METHOD PUBLIC initJntPos : BOOL
VAR_INPUT
END_VAR
m_lastLinkEncoder :=m_motorInputs.m_linkEncoder;
m_linkEncCycles:=0;
m_curLinkPos :=linkEnc2Pos();
m_initLinkPos:=m_curLinkPos;
m_initMotorEnc :=m_motorInputs.m_motorEncoder;
m_curMotorPos:=motorEnc2Pos();
m_curJntPos := m_curMotorPos;
m_cmdJntPos :=m_curJntPos;	
m_lastJntPos :=m_curJntPos;
m_lastLinkPos := m_curLinkPos;

// filter init
m_jntVelLpf.init(1, g_curJntVelLpfCutoffFreq, g_armCtrlFreq);
m_linkVelLpf.init(1, g_curJntVelLpfCutoffFreq, g_armCtrlFreq);
END_METHOD

// reset the initial joint position with input value
METHOD PUBLIC initJntPosReset : BOOL
VAR_INPUT
	i_initLinkPos:LREAL;
END_VAR
m_initLinkPos:=i_initLinkPos;
m_initMotorEnc :=m_motorInputs.m_motorEncoder;
m_curMotorPos:=motorEnc2Pos();
m_curJntPos := m_curMotorPos;
m_cmdJntPos :=m_curJntPos;	
m_lastJntPos :=m_curJntPos;
m_lastLinkPos := m_curLinkPos;

// filter init
m_jntVelLpf.init(1, g_curJntVelLpfCutoffFreq, g_armCtrlFreq);
m_linkVelLpf.init(1, g_curJntVelLpfCutoffFreq, g_armCtrlFreq);
END_METHOD

PROPERTY initLinkPos : lreal
GET
initLinkPos:=m_initLinkPos;
END_GET
SET
m_initLinkPos:=initLinkPos;
END_SET
END_PROPERTY

METHOD PUBLIC isEnabled : BOOL
VAR_INPUT
END_VAR
isEnabled :=(DriverStatusWord_OP = m_motorInputs.m_statusWord);
END_METHOD

PROPERTY jntPos : LREAL
GET
jntPos := m_curJntPos;
END_GET
END_PROPERTY

PROPERTY jntTrq : LREAL
GET
jntTrq:=m_curJntTrq;
END_GET
END_PROPERTY

PROPERTY jntVel : LREAL
GET
jntVel := m_curJntVel;
END_GET
END_PROPERTY

METHOD PROTECTED linkEnc2Pos : LREAL
VAR_INPUT
END_VAR
VAR
	incLinkPos :LREAL;
	newLinkEnc :DINT;
END_VAR
// cycle check
IF 1=m_multiCycles THEN
	IF (m_motorInputs.m_linkEncoder - m_lastLinkEncoder)*m_linkEncoderDir < -m_linkEncoderRes/2 THEN
		m_linkEncCycles :=m_linkEncCycles+1;
	ELSIF (m_motorInputs.m_linkEncoder - m_lastLinkEncoder)*m_linkEncoderDir > m_linkEncoderRes/2 THEN
		m_linkEncCycles :=m_linkEncCycles-1;
	END_IF
END_IF
m_lastLinkEncoder:=m_motorInputs.m_linkEncoder;

// convert link encoder if joint cross zero
newLinkEnc := m_motorInputs.m_linkEncoder;
IF 1=m_linkEncZeroCross AND 0 = m_multiCycles THEN
	IF 1=m_linkEncoderDir AND m_motorInputs.m_linkEncoder < m_minLinkEncoder THEN
		newLinkEnc := m_motorInputs.m_linkEncoder + m_linkEncoderRes;
	ELSIF -1=m_linkEncoderDir AND m_motorInputs.m_linkEncoder < m_maxLinkEncoder THEN
		newLinkEnc := m_motorInputs.m_linkEncoder + m_linkEncoderRes;
	END_IF
END_IF

// motion from calibrated points
incLinkPos := (newLinkEnc-m_caliLinkEncoder)*m_linkEnc2PosRatio;

// absolute joint position
linkEnc2Pos := incLinkPos + m_linkEncCaliJntPos + 2*PI* m_linkEncCycles;
END_METHOD

PROPERTY PUBLIC linkPos : LREAL
GET
linkPos:=m_curLinkPos;
END_GET
END_PROPERTY

METHOD PROTECTED motorEnc2Pos : LREAL
VAR_INPUT
END_VAR
motorEnc2Pos:= (m_motorInputs.m_motorEncoder-m_initMotorEnc)* m_motorEnc2PosRatio +m_initLinkPos;
END_METHOD

PROPERTY PUBLIC motorPos : LREAL
GET
motorPos := m_curMotorPos;
END_GET
END_PROPERTY

METHOD PROTECTED motorPos2Enc : DINT
VAR_INPUT
	i_jntPos :LREAL;
END_VAR

VAR
END_VAR
motorPos2Enc := LREAL_TO_DINT((i_jntPos-m_initLinkPos)/m_motorEnc2PosRatio + m_initMotorEnc);
END_METHOD

PROPERTY rawCurrent : LREAL
GET
rawCurrent := m_rawCurrent;
END_GET
END_PROPERTY

METHOD PUBLIC updateCmds : BOOL
VAR_INPUT
	i_opMode : E_DriverOPMode;
	i_cmdPos :LREAL;
	i_cmdTrq :LREAL;
END_VAR
VAR
	filtCmdTrq :LREAL;
END_VAR
m_motorOutputs.m_opMode:=INT_TO_SINT( i_opMode);
// pos mode
IF i_opMode = DriverOPMode_Pos THEN
	m_motorOutputs.m_cmdCurrent:=0;
	m_cmdTrqLpf.reset();
//	i_cmdPos:=LIMIT(m_minJntPos, i_cmdPos, m_maxJntPos);
	m_motorOutputs.m_cmdMotorEncoder :=motorPos2Enc(i_cmdPos);
ELSIF i_opMode = DriverOPMode_Trq THEN
	filtCmdTrq:=m_cmdTrqLpf.run(i_cmdTrq);
	m_motorOutputs.m_cmdCurrent:=LREAL_TO_DINT(LIMIT(-m_maxCurrent, filtCmdTrq*m_trq2CurrentRatio,m_maxCurrent));
	m_motorOutputs.m_cmdMotorEncoder :=m_motorInputs.m_motorEncoder; 
END_IF
m_cmdCurrent:=m_motorOutputs.m_cmdCurrent;
END_METHOD

METHOD PUBLIC updateStatus : BOOL
VAR_INPUT
END_VAR
// compute joint position
m_curLinkPos:= linkEnc2Pos();
m_curMotorPos:=motorEnc2Pos();
m_curJntPos := m_curMotorPos;

// compute joint velocity
m_curJntVel:= (m_curJntPos-m_lastJntPos)/m_cycleTime;
m_curJntVel := m_jntVelLpf.run(m_curJntVel);
m_lastJntPos :=m_curJntPos;

// compute link velocity
m_curLinkVel := (m_curLinkPos-m_lastLinkPos)/m_cycleTime;
m_curLinkVel := m_linkVelLpf.run(m_curLinkVel);
m_lastLinkPos := m_curLinkPos;

//compute joint acceleration
m_curJntAcc:=(m_curJntVel-m_lastJntVel)/m_cycleTime;
m_curJntAcc := m_jntAccLpf.run(m_curJntAcc);
m_lastJntVel:=m_curJntVel;

//compute link acceleration
m_curLinkAcc:=(m_curLinkVel-m_lastLinkVel)/m_cycleTime;
m_curLinkAcc := m_linkAccLpf.run(m_curLinkAcc);
m_lastLinkVel:=m_curLinkVel;

// current and torque
m_rawCurrent := m_motorInputs.m_current;
m_filtCurrent := m_curTrqLpf.run(m_rawCurrent);
m_curJntTrq := m_filtCurrent * m_current2TrqRatio;
END_METHOD

END_FUNCTION_BLOCK

// ---- FBs_RobotDynamics/FB_MasterFriciton.TcPOU
FUNCTION_BLOCK FB_MasterFriciton
VAR_INPUT
END_VAR
VAR_OUTPUT
END_VAR
VAR
	// joint friction compensation scale
	m_frictionCompScale :Vec7d :=[0.7, 0.5, 0.5, 0.0, 0.7, 0.7, 0.7];
	
	// joint velocity threshold for coulomb friction transition
	m_cFrictionVelThres : LREAL := 5.0 * g_deg2Rad;
	
	// arm index
	m_armIdx: INT ;
	
	// joint coulomb friction parameters: friction = a * gravityTrq + b;
	m_frictionParamA : Vec7d := g_zeroVec7d;
	m_frictionParamB : Vec7d := g_zeroVec7d;
	
	// joint damping
	m_jntDamp :Vec7d := g_zeroVec7d;
	
	// max joint friciton 
	m_maxFriction :Vec7d;
	

END_VAR

METHOD init : BOOL
VAR_INPUT
	i_armIdx :INT;
END_VAR

VAR
	i:int;
END_VAR
m_armIdx := i_armIdx;

m_frictionParamA := g_zeroVec7d;
m_frictionParamB := g_zeroVec7d;
m_jntDamp := g_zeroVec7d;
m_maxFriction := GVL_ArmDynamics.g_maxJntFriction;

FOR i:=1 TO 7 DO
	m_frictionParamA[i] := GVL_ArmDynamics.g_jntFrictionParam[m_armIdx, 2*i-1];
	m_frictionParamB[i] := GVL_ArmDynamics.g_jntFrictionParam[m_armIdx, 2*i];
END_FOR
END_METHOD

METHOD run : vec7d
VAR_IN_OUT CONSTANT
	// joint gravity torque
	i_jntGravity :Vec7d;
	
	// joint velocity
	i_jntVel :Vec7d;
END_VAR

VAR
	i:INT;
	transitScale:LREAL;
	cFriction, dFriction :LREAL;
END_VAR
FOR i:=1 TO g_mJntNum DO
	transitScale := LIMIT(0, ABS(i_jntVel[i]/m_cFrictionVelThres),1);
	cFriction:=m_frictionParamA[i]*ABS(i_jntGravity[i])+m_frictionParamB[i];
	cFriction:= transitScale * sign(i_jntVel[i]) * cFriction;
	
	dFriction:= i_jntVel[i] * m_jntDamp[i];
	
	run[i] := LIMIT(-m_maxFriction[i], m_frictionCompScale[i] * (cFriction+dFriction) ,m_maxFriction[i]);
END_FOR
END_METHOD

END_FUNCTION_BLOCK

// ---- FBs_Robots/FB_CartJoint.TcPOU
FUNCTION_BLOCK FB_CartJoint EXTENDS FB_JointBase
VAR_INPUT
END_VAR
VAR_OUTPUT
END_VAR
VAR
END_VAR

METHOD PUBLIC init : BOOL
VAR_INPUT
	i_jntIdx :INT;
	i_controlCycleTime :LREAL;
END_VAR
m_cycleTime := i_controlCycleTime;

// hardware parameters
m_motorEncoderRes :=GVL_CartJointParameters.g_incEncoderRes[i_jntIdx];
m_linkEncoderRes :=GVL_CartJointParameters.g_absEncoderRes[i_jntIdx];
m_motorReduction :=GVL_CartJointParameters.g_motorReduction[i_jntIdx];
m_linkEncoderReduction :=GVL_CartJointParameters.g_absEncoderReduction[i_jntIdx];
m_trqConst :=GVL_CartJointParameters.g_motorTrqConst[i_jntIdx];
m_maxCurrent :=GVL_CartJointParameters.g_motorMaxCurrent[i_jntIdx];
m_motorDir :=GVL_CartJointParameters.g_motorDir[i_jntIdx];								
m_linkEncoderDir :=GVL_CartJointParameters.g_asbEncoderDir[i_jntIdx];
m_minJntPos	:=GVL_CartJointParameters.g_minJntPos[i_jntIdx];
m_maxJntPos	:=GVL_CartJointParameters.g_maxJntPos[i_jntIdx];

//link encoder calibartion data
m_minLinkEncoder :=GVL_CartJointCaliData.g_minLinkEncoder[i_jntIdx] - m_linkEncoderDir*GVL_CartJointCaliData.g_linkEncLimitBuffer; // expand limit
m_maxLinkEncoder :=GVL_CartJointCaliData.g_maxLinkEncoder[ i_jntIdx] + m_linkEncoderDir*GVL_CartJointCaliData.g_linkEncLimitBuffer; // expand limit
m_caliLinkEncoder :=GVL_CartJointCaliData.g_caliLinkEncoder[i_jntIdx];
m_linkEncCaliJntPos :=GVL_CartJointCaliData.g_linkEncCaliJntPos[i_jntIdx];
m_linkEncZeroCross :=GVL_CartJointCaliData.g_linkEncZeroCross[i_jntIdx];
m_multiCycles :=GVL_CartJointCaliData.g_multipleCyclesJoint[i_jntIdx];

// convert cali link encoder if joint cross zero
IF 1=m_linkEncZeroCross THEN
	IF 1=m_linkEncoderDir AND m_caliLinkEncoder < m_minLinkEncoder THEN
		m_caliLinkEncoder := GVL_CartJointCaliData.g_caliLinkEncoder[i_jntIdx] + m_linkEncoderRes;
	ELSIF -1=m_linkEncoderDir AND m_caliLinkEncoder < m_maxLinkEncoder THEN
		m_caliLinkEncoder := GVL_CartJointCaliData.g_caliLinkEncoder[i_jntIdx] + m_linkEncoderRes;
	END_IF
END_IF

// macro data
m_trq2CurrentRatio:=m_motorDir * 1000.0/(m_trqConst*m_motorReduction);
m_current2TrqRatio:=m_motorDir * (m_trqConst*m_motorReduction)/1000.0;
m_linkEnc2PosRatio := 2*PI*m_linkEncoderDir/(m_linkEncoderReduction*m_linkEncoderRes);
m_motorEnc2PosRatio := 2*PI * m_motorDir/(m_motorReduction * m_motorEncoderRes);

// motor data init
m_curJntVel:=0;
m_curJntTrq :=0;
m_rawCurrent :=0;
m_filtCurrent :=0;
m_cmdJntVel :=0.0;
m_cmdJntTrq :=0.0;
m_cmdCurrent := 0.0;

// filter init
m_cmdTrqLpf.init(1, g_cmdJntTrqLpfCutoffFreq, g_cartCtrlFreq);
m_curTrqLpf.init(1, g_curJntTrqLpfCutoffFreq, g_cartCtrlFreq);
m_jntVelLpf.init(1, g_curJntVelLpfCutoffFreq, g_cartCtrlFreq);
m_linkVelLpf.init(1, g_curJntVelLpfCutoffFreq, g_cartCtrlFreq);
m_jntAccLpf.init(1, g_curJntVelLpfCutoffFreq*0.2, g_armCtrlFreq); 
m_linkAccLpf.init(1, g_curJntVelLpfCutoffFreq*0.2, g_armCtrlFreq); 


// driver init value
m_motorOutputs.m_controlWord:=DriverCtrlWord_INIT;
m_motorOutputs.m_opMode:=INT_TO_SINT(DriverOPMode_Pos);
m_motorOutputs.m_cmdCurrent:=0;
m_motorOutputs.m_cmdMotorEncoder:=m_motorInputs.m_motorEncoder;
END_METHOD

END_FUNCTION_BLOCK

// ---- FBs_Robots/FB_MasterCart.TcPOU
FUNCTION_BLOCK FB_MasterCart
VAR
	//  IO and check
	m_endoScopePedalIO AT%I* :BOOL;
	m_endoScopeIOCheck :FB_IOCheck;
	
	m_clutchPedalIO AT%I* :BOOL;
	m_clutchIOCheck :FB_IOCheck;
	
	m_surgonHeadInIO AT%I* :BOOL;
	m_headInCheck:FB_IOCheck;
	
	m_armSwitchIO AT%I* :BOOL;
	m_armSwitchCheck:FB_IOToggleCheck;
	
	m_electricCutLeft AT %I* :BOOL;
	m_electricCutLeftAllow AT %I* :BOOL;
	
	m_electricCutRight AT %I* :BOOL;
	m_electricCutRightAllow AT %I* :BOOL;
	
	m_electricCoagulLeft AT %I* :BOOL;
	m_electricCoagulLeftAllow AT %I* :BOOL;
	
	m_electricCoagulRight AT %I* :BOOL;
	m_electricCoagulRightAllow AT %I* :BOOL;
	
	m_elecKnifeCtrlWord AT %Q* :DINT;
	
	// cart status
	m_cartStatus  : ST_CartStatus;
	
	// cart joints
	// [monitor lift, monitor rotate, armset, pedal]
	m_cartJoints:ARRAY[1..4] OF FB_CartJoint;
	
	// cart joint motion control IO
	//[monitor_up, monitor_down, monitor_cwRotate, monitor_ccwRotate, armset_up, armset_down, pedal_in, pedal_out]
	m_cartJointCtrlIO AT%I* :ARRAY[1..8] OF BOOL ;
	m_cartJointCtrlIOCheck :ARRAY[1..8] OF FB_IOCheck;
	
	//electrotome control io
	m_electricCutLeftOn :BOOL;
	m_electricCutRightOn :BOOL;
	m_electricCoagulLeftOn : BOOL;
	m_electricCoagulRightOn : BOOL;
	//Triggering several energies at once
	m_eleCtrlState : UINT;
	//The type of instrument energy of the master hand corresponding to the slave hand
	m_energyType :ARRAY[1..g_mArmNum] OF UINT :=[2(0)];
	
	// cart joint control data
	m_jntEnableCounts:Vec4i ;
	m_jntDisableCounts:Vec4i ;
	m_jntEnableCountsThres:INT:=500;
	m_jntCmdMotionDir :Vec4i;
	m_cmdJntTrq :Vec4d;
	m_cmdJntPos :Vec4d;
	m_cmdJntVel :Vec4d;
	m_jntEnableFlag :Vec4b;
	
	//cart ergonomic adjust data
	m_UIData : ST_CartUIData;
	m_carInMotion : INT; // 0:  no mition, 1: mamual adjust, 2: ergonomic adjust
	m_jntSoftwareLimit :ARRAY [1..4] OF LREAL := [0.001, 1*g_deg2Rad, 0.001, 0.001];
	m_cmdArrival : Vec4b;
	
	// cart joint status data
	m_curMotorPos :Vec4d;
	m_curLinkPos :Vec4d;
	m_curJntPos :Vec4d;
	m_curJntVel :Vec4d;
	m_curJntTrq :Vec4d;
	m_rawJntCurrent :Vec4d;
	m_filtJntCurrent :Vec4d;
	m_cmdJntCurrent : Vec4d;

END_VAR

METHOD eleKnifeCtrl : DINT
VAR_IN_OUT CONSTANT
	m_armState:ARRAY[1..g_mArmNum] OF E_masterArmState ;
	m_teleSlaveArmIdx :ARRAY[1..g_mArmNum] OF E_MatchedSlaveArmIdx;
	m_instruStauts: ARRAY[1..g_sArmNum] OF ST_InstruStatus;
END_VAR
//Foot trigger check
m_electricCutLeftOn := m_electricCutLeft AND m_electricCutLeftAllow AND m_armState[1] = MasterArmState_MasterSlave ;
m_electricCutRightOn := m_electricCutRight AND m_electricCutRightAllow AND m_armState[2] = MasterArmState_MasterSlave ;
m_electricCoagulLeftOn := m_electricCoagulLeft AND m_electricCoagulLeftAllow AND m_armState[1] = MasterArmState_MasterSlave ;
m_electricCoagulRightOn := m_electricCoagulRight AND m_electricCoagulRightAllow AND m_armState[2] = MasterArmState_MasterSlave ;

//You cannot excite two energies at the same time
m_eleCtrlState := BOOL_TO_UINT(m_electricCutLeftOn) + BOOL_TO_UINT(m_electricCutRightOn)
										 + BOOL_TO_UINT(m_electricCoagulLeftOn) + BOOL_TO_UINT(m_electricCoagulRightOn);

IF m_teleSlaveArmIdx[1] > 0 THEN
	m_energyType[1] := m_instruStauts[m_teleSlaveArmIdx[1]].m_energyType;
	m_energyType[2] := m_instruStauts[m_teleSlaveArmIdx[2]].m_energyType;
END_IF

IF m_eleCtrlState = 1 THEN
	IF (m_electricCutLeftOn AND  m_energyType[1] = InstruType_isMonopole) OR (m_electricCutRightOn AND  m_energyType[2] = InstruType_isMonopole) THEN
		eleKnifeCtrl := EnergyCtrlWord_isMonopoleCut;
	ELSIF (m_electricCoagulLeftOn AND m_energyType[1] = InstruType_isMonopole) OR (m_electricCoagulRightOn AND  m_energyType[2] = InstruType_isMonopole) THEN
		eleKnifeCtrl := EnergyCtrlWord_isMonopoleCoagul;
	ELSIF (m_electricCoagulLeftOn AND m_energyType[1] = InstruType_isBipolar) OR (m_electricCoagulRightOn AND  m_energyType[2] = InstruType_isBipolar) THEN
		eleKnifeCtrl := EnergyCtrlWord_isBipolarCoagul;
	ELSIF (m_electricCutLeftOn AND m_energyType[1] = InstruType_isUltraKnife) OR (m_electricCutRightOn AND  m_energyType[2] = InstruType_isUltraKnife) THEN
		eleKnifeCtrl := EnergyCtrlWord_isUltraMin;
	ELSIF (m_electricCoagulLeftOn AND m_energyType[1] = InstruType_isUltraKnife) OR (m_electricCoagulRightOn AND  m_energyType[2] = InstruType_isUltraKnife) THEN
		eleKnifeCtrl := EnergyCtrlWord_isUltraMax;
		
	ELSE
		eleKnifeCtrl := EnergyCtrlWord_NoOutput;
	END_IF
ELSE
	eleKnifeCtrl := EnergyCtrlWord_NoOutput;
END_IF
END_METHOD

METHOD ergonomicAdjust : INT
VAR_INPUT
END_VAR
VAR
	i : INT;
	err:Vec4d;
END_VAR
vecSub(m_UIData.m_cmdJntPos,m_curJntPos, err);
ergonomicAdjust := 2;
//only update command after joints is truly enabled
FOR i := 1 TO 4 DO
	IF m_jntEnableFlag[i] AND m_cartJoints[i].isEnabled() AND m_jntEnableCounts[i]>= m_jntEnableCountsThres THEN
		m_cmdJntVel[i]:=sign(m_UIData.m_cmdJntPos[i]-m_cartJoints[i].jntPos)*(GVL_CartJointParameters.g_jntCtrlMotionVel[i]);
		IF ABS(err[i]) < m_jntSoftwareLimit[i]/3 THEN
			m_cmdJntVel[i]:=0;
		END_IF
		m_cmdJntPos[i] := LIMIT(GVL_CartJointParameters.g_minJntPos[i] + m_jntSoftwareLimit[i],  m_cmdJntPos[i] + m_cmdJntVel[i]*g_cartCtrlCycleTime, GVL_CartJointParameters.g_maxJntPos[i] - m_jntSoftwareLimit[i]);
	
	ELSE
		m_cmdJntVel[i]:=0;
		m_cmdJntPos[i] := m_cartJoints[i].jntPos;
	END_IF	
END_FOR
END_METHOD

METHOD PUBLIC getStatus : BOOL
VAR_IN_OUT
	// cart status data
	r_cartStatus :ST_CartStatus;
	
	// cart joint data
	r_cartJointData :ST_CartJointData;
	
END_VAR
r_cartStatus := m_cartStatus;


// current joint data
r_cartJointData.m_curMotorPos:=m_curMotorPos;
r_cartJointData.m_curLinkPos:=m_curLinkPos;
r_cartJointData.m_curJntPos:=m_curJntPos;
r_cartJointData.m_curJntVel:=m_curJntVel;
r_cartJointData.m_curJntTrq:=m_curJntVel;
r_cartJointData.m_rawJntCurrent:=m_rawJntCurrent;
r_cartJointData.m_filtJntCurrent:=m_filtJntCurrent;

// command joint data
r_cartJointData.m_cmdJntPos:=m_cmdJntPos;
r_cartJointData.m_cmdJntVel:=m_cmdJntVel;
r_cartJointData.m_cmdJntTrq:=m_cmdJntTrq;
r_cartJointData.m_cmdJntCurrent:=m_cmdJntCurrent;
END_METHOD

METHOD PUBLIC init : BOOL
VAR_INPUT
END_VAR
VAR
	i:INT;
	initLinkPos :LREAl;
END_VAR
// joint init
FOR i:=1 TO 4 DO
	m_cartJoints[i].init(i,g_cartCtrlCycleTime);
	m_cartJoints[i].initJntPos();
END_FOR

// motor and link encoder of  monitor rotation are on different  joints
// transfer monitor angle from link side to motor side
initLinkPos:= monitorAngLink2Motor(m_cartJoints[2].initLinkPos);
m_cartJoints[2].initJntPosReset(initLinkPos);

// init commands
FOR i:=1 TO 4 DO
	m_jntEnableCounts[i]:=0;
	m_jntDisableCounts[i]:=0;
	m_jntEnableFlag[i]:=FALSE;
	m_jntCmdMotionDir[i]:=0;
	m_cmdJntTrq[i]:=0;
	m_cmdJntVel[i]:=0;
	m_cmdJntPos[i]:=m_cartJoints[i].jntPos;
END_FOR

m_cartStatus.m_initFlag :=true;
END_METHOD

METHOD manualAdjust : INT
VAR_INPUT
END_VAR
VAR
	i : INT;
END_VAR
// update joint command positon
manualAdjust := 1;
//only update command after joints is truly enabled
FOR i := 1 TO 4 DO
	IF  m_jntEnableFlag[i] AND m_cartJoints[i].isEnabled() AND m_jntEnableCounts[i]>= m_jntEnableCountsThres THEN
		//  update command joint velocity
		m_cmdJntVel[i]:=m_jntCmdMotionDir[i]*GVL_CartJointParameters.g_jntCtrlMotionVel[i];
		
		// limit handle
		IF (m_cmdJntPos[i]> GVL_CartJointParameters.g_maxJntPos[i] - m_jntSoftwareLimit[i] AND m_cmdJntVel[i] >0 ) OR 
				(m_cmdJntPos[i]< GVL_CartJointParameters.g_minJntPos[i] + m_jntSoftwareLimit[i] AND m_cmdJntVel[i] <0 )  THEN
				m_cmdJntVel[i] := 0.0;
		END_IF
		m_cmdJntPos[i]:= m_cmdJntPos[i]+ m_cmdJntVel[i]*g_cartCtrlCycleTime;
	ELSE
		m_cmdJntVel[i]:=0;
		m_cmdJntPos[i] := m_cartJoints[i].jntPos;
	END_IF
END_FOR
END_METHOD

// TODO
METHOD PROTECTED monitorAngLink2Image : LREAL
VAR_INPUT
	i_linkPos:LREAL;
END_VAR
VAR
	A,B,C,D,E,F,G,H,I,X0,X1,X2,X3,X4,X5,X6,X7,X8,X9,X10,X11,X12,Z0:LREAL;	
END_VAR

X0:=i_linkPos;  //监视器旋转

A:=227; B:=216; C:=159.285; D:=150.297; E:=195; F:=130; G:=137; H:=40; I:=99;
X4:=ATAN(H/I); X5:=ATAN(F/G);
X8:=SQRT(F*F+G*G);
X12:=sqrt(H*H+I*I);
X9:=sqrt(E*E+X12*X12-2*E*X12*cos(X0));
X6:=acos((B*B+X8*X8-X9*X9)/(2*B*X8));
X10:=acos((B*B+X9*X9-X8*X8)/(2*B*X9));
X11:=acos((X9*X9+X12*X12-E*E)/(2*X9*X12));
X7:=X10+X11;
X2:=X5-X6;
X3:=pi-X7+X2;
X1:=X3-X4;

monitorAngLink2Image:=X1;
END_METHOD

// TODO
METHOD PROTECTED monitorAngLink2Motor : LREAL
VAR_INPUT
	i_linkPos:LREAL;
END_VAR
VAR
	A,B,C,D,E,F,G,H,I,X0,X1,X2,X3,X4,X5,X6,X7,X8,X9,X10,X11,X12,Z0:LREAL;	
END_VAR

X0:=i_linkPos;  //监视器旋转

A:=227; B:=216; C:=159.285; D:=150.297; E:=195; F:=130; G:=137; H:=40; I:=99;
X4:=ATAN(H/I); X5:=ATAN(F/G);
X8:=SQRT(F*F+G*G);
X12:=sqrt(H*H+I*I);
X9:=sqrt(E*E+X12*X12-2*E*X12*cos(X0));
X6:=acos((B*B+X8*X8-X9*X9)/(2*B*X8));
X10:=acos((B*B+X9*X9-X8*X8)/(2*B*X9));
X11:=acos((X9*X9+X12*X12-E*E)/(2*X9*X12));
X7:=X10+X11;
X2:=X5-X6;
X3:=pi-X7+X2;
X1:=X3-X4;

monitorAngLink2Motor:=X2;
END_METHOD

//TODO
METHOD PROTECTED monitorAngMotor2Link : LREAL
VAR_INPUT
	i_motorPos:LREAL;
END_VAR
VAR
	A,B,C,D,E,F,G,H,I,X0,X1,X2,X3,X4,X5,X6,X7,X8,X9,X10,X11,X12,Z0:LREAL;	
END_VAR
X2:=i_motorPos;

A:=227; B:=216; C:=159.285; D:=150.297; E:=195; F:=130; G:=137; H:=40; I:=99;
X5:=atan(F/G);
X6:=X5-X2;
X8:=sqrt(F*F+G*G);
X9:=sqrt(B*B+X8*X8-2*B*X8*cos(X6));
X12:=SQRT(H*H+I*I);
X0:=ACOS((E*E+X12*X12-X9*X9)/(2*E*X12));

monitorAngMotor2Link:=X0;
END_METHOD

METHOD reachUITargetCheck : bool
VAR
	i :INT;
	err:Vec4d;
END_VAR
vecSub(m_UIData.m_cmdJntPos,m_curJntPos, err);

// joint error check
FOR i:=1 TO 4 DO 
	m_cmdArrival[i] :=  ABS(err[i]) < m_jntSoftwareLimit[i]/2;
END_FOR
END_METHOD

METHOD PUBLIC run : BOOL
VAR_IN_OUT CONSTANT
	i_cartUIData : ST_CartUIData;
END_VAR
VAR
	i:INT;
END_VAR
// update IO signals
updateIO(i_cartUIData);

// update cart status
updateStatus();

// update controller and command
updateCmds();

// send command to joint driver
FOR i:=1 TO 4 DO
	// joint enable
	IF m_jntEnableFlag[i] AND NOT(SafetyCheck.m_safetyCheckData.m_cartErrFlag[i]) AND MasterArmControl.m_masterStatus.m_armState[1] <> MasterArmState_MasterSlave 
								AND MasterArmControl.m_masterStatus.m_armState[2] <> MasterArmState_MasterSlave THEN
		m_cartJoints[i].enable();
	ELSE
		m_cartJoints[i].disable();
	END_IF
	
	// set command position
	m_cartJoints[i].updateCmds(DriverOPMode_Pos,m_cmdJntPos[i],m_cmdJntTrq[i]);
END_FOR
END_METHOD

PROPERTY status : ST_CartStatus
GET
status := m_cartStatus;
END_GET
END_PROPERTY

METHOD PROTECTED updateCmds : BOOL
VAR_INPUT
END_VAR
VAR
	i:INT;
	
END_VAR
IF (m_jntCmdMotionDir[1] <>0 OR m_jntCmdMotionDir[2]<>0 OR m_jntCmdMotionDir[3] <>0 OR m_jntCmdMotionDir[4] <>0) AND m_carInMotion <> 2 THEN
	m_carInMotion := manualAdjust();
ELSIF (m_UIData.m_ergonomicCrl.m_recovErgonEnable OR m_UIData.m_ergonomicCrl.m_cancelRecovErgonEnable) AND m_carInMotion <> 1 THEN
	m_carInMotion := ergonomicAdjust();
ELSE
	m_carInMotion := 0;
END_IF

reachUITargetCheck();
IF m_cmdArrival[1] AND m_cmdArrival[2] AND m_cmdArrival[3] AND m_cmdArrival[4] THEN
	IF m_UIData.m_ergonomicCrl.m_recovErgonEnable THEN
		m_cartStatus.m_cancelErgonAdjustArrival := FALSE;
		m_cartStatus.m_ergonAdjustArrival := TRUE;
	END_IF
	IF m_UIData.m_ergonomicCrl.m_cancelRecovErgonEnable THEN
		m_cartStatus.m_ergonAdjustArrival := FALSE;
		m_cartStatus.m_cancelErgonAdjustArrival := TRUE;
	END_IF
ELSE
	m_cartStatus.m_ergonAdjustArrival := FALSE;
	IF m_UIData.m_ergonomicCrl.m_recovErgonEnable THEN
		m_cartStatus.m_cancelErgonAdjustArrival := FALSE;
	END_IF
END_IF
END_METHOD

METHOD PROTECTED updateIO : BOOL
VAR_INPUT
	i_cartUIData : ST_CartUIData;
END_VAR
VAR
	i:INT;
	idxOffset:INT;
END_VAR
// updata IO signals
m_cartStatus.m_clutchSwitch:= m_clutchIOCheck.check(m_clutchPedalIO);
m_cartStatus.m_endoscopeSwitch := m_endoScopeIOCheck.check(m_endoScopePedalIO);
m_cartStatus.m_surgonReady := m_headInCheck.check(m_surgonHeadInIO);
m_cartStatus.m_armSwitch :=m_armSwitchCheck.check(m_armSwitchIO);
m_UIData := i_cartUIData;

//updata Electrotome control
m_elecKnifeCtrlWord := eleKnifeCtrl(MasterArmControl.m_masterStatus.m_armState , MasterArmControl.m_masterStatus.m_teleSlaveArmIdx , MasterArmControl.m_masterInputDataPool.m_slaveStatus.m_instruStauts );

//updata pedal hover and pedal trigger
m_cartStatus. m_pedalHover[1] := m_electricCutLeftAllow OR m_electricCoagulLeftAllow;
m_cartStatus. m_pedalHover[2] := m_electricCutRightAllow OR m_electricCoagulRightAllow;
IF m_electricCutLeftOn AND m_eleCtrlState = 1 THEN
	m_cartStatus.m_electricKnifePedalTrigger[1] := 1;
ELSIF m_electricCoagulLeftOn AND m_eleCtrlState = 1 THEN
	m_cartStatus.m_electricKnifePedalTrigger[1] := 2;
ELSE
	m_cartStatus.m_electricKnifePedalTrigger[1] := 0;
END_IF

IF m_electricCutRightOn AND m_eleCtrlState = 1 THEN
	m_cartStatus.m_electricKnifePedalTrigger[2] := 1;
ELSIF m_electricCoagulRightOn AND m_eleCtrlState = 1 THEN
	m_cartStatus.m_electricKnifePedalTrigger[2] := 2;
ELSE
	m_cartStatus.m_electricKnifePedalTrigger[2] := 0;
END_IF

//update cart joint control switch
FOR i:=1 TO 4 DO 
	idxOffset:= 2*(i-1);
	IF m_cartJointCtrlIOCheck[1+idxOffset].check(m_cartJointCtrlIO[1+idxOffset]) THEN
		m_jntCmdMotionDir[i]:=1;
	ELSIF  m_cartJointCtrlIOCheck[2+idxOffset].check(m_cartJointCtrlIO[2+idxOffset]) THEN
		m_jntCmdMotionDir[i]:=-1;
	ELSE
		m_jntCmdMotionDir[i]:=0;
	END_IF
END_FOR


// if console is already in motion, only check the currently moving joint
IF m_cartStatus.m_consoleInAdjust THEN
	FOR i:=1 TO 4 DO
		IF NOT(m_cartJoints[i].isEnabled()) THEN
			m_jntCmdMotionDir[i] := 0;
		END_IF
	END_FOR
END_IF


// update joint enable flag
FOR i:= 1 TO 4 DO
	IF m_jntCmdMotionDir[i] <> 0 OR m_UIData.m_ergonomicCrl.m_recovErgonEnable OR m_UIData.m_ergonomicCrl.m_cancelRecovErgonEnable THEN
		m_jntEnableFlag[i] := TRUE;
		m_jntEnableCounts[i]:= LIMIT(0, m_jntEnableCounts[i]+1, m_jntEnableCountsThres);
		m_jntDisableCounts[i]:=m_jntEnableCountsThres;
	ELSE
		m_jntEnableCounts[i]:=0;
		m_jntDisableCounts[i]:= LIMIT(0, m_jntDisableCounts[i]-1, m_jntEnableCountsThres);
		m_jntEnableFlag[i] :=m_jntDisableCounts[i]>0; 
	END_IF
END_FOR

// Do not adjust during master-slave control
IF MasterArmControl.m_masterStatus.m_armState[1] = MasterArmState_MasterSlave OR MasterArmControl.m_masterStatus.m_armState[1] = MasterArmState_Endoscope OR
	MasterArmControl.m_masterStatus.m_armState[2] = MasterArmState_MasterSlave OR MasterArmControl.m_masterStatus.m_armState[2] = MasterArmState_Endoscope  THEN
	m_jntCmdMotionDir := g_zeroVec4i;
END_IF
END_METHOD

METHOD PROTECTED updateStatus : BOOL
VAR_INPUT
END_VAR
VAR
	i:INT;
END_VAR
// update cart joints status
FOR i:=1  TO 4 DO
	m_cartJoints[i].updateStatus();
END_FOR

// get joint data
FOR i:=1 TO 4 DO
	m_curMotorPos[i]:=m_cartJoints[i].motorPos;
	m_curLinkPos[i]:=m_cartJoints[i].linkPos;
	m_curJntPos[i]:=m_cartJoints[i].jntPos;
	m_curJntVel[i]:=m_cartJoints[i].jntVel;
	m_curJntTrq[i]:=m_cartJoints[i].jntTrq;
	m_rawJntCurrent[i]:=m_cartJoints[i].rawCurrent;
	m_filtJntCurrent[i]:=m_cartJoints[i].filtCurrent;
	m_cmdJntCurrent[i]:=m_cartJoints[i].cmdCurrent;
END_FOR 

// transfer monitor angle from link side to motor side
m_curLinkPos[2]:= monitorAngLink2Motor(m_cartJoints[2].linkPos);

// get monitor angle
m_cartStatus.m_monitorAngle:= monitorAngLink2Image(m_cartJoints[2].linkPos);

// check if cart in motion
m_cartStatus.m_consoleInAdjust:=FALSE;
FOR i:=1 TO 4 DO
	IF m_cartJoints[i].isEnabled() THEN
		m_cartStatus.m_consoleInAdjust:=TRUE;
		EXIT;
	END_IF
END_FOR

// check if monitor in motion
m_cartStatus.m_monitorInAdjust:=m_cartJoints[2].isEnabled();

// check if cart in manual adjustment
m_cartStatus.m_consoleInManualAdjust := FALSE;
FOR i:=1 TO 4 DO
	IF m_jntCmdMotionDir[i] <> 0 AND m_cartJoints[i].isEnabled() THEN
		m_cartStatus.m_consoleInManualAdjust := TRUE;
		EXIT;
	END_IF
END_FOR
END_METHOD

END_FUNCTION_BLOCK

// ---- Mains/MasterArmControl.TcPOU
PROGRAM MasterArmControl
VAR
	// slave robot data, input from slave controller box
	m_slaveRobotData AT %I* : MSCommu_slaveStatus;
	
	// all data from other tasks and controller 
	m_masterInputDataPool : ST_MasterInputDataPool;
	
	// master robot information, including arm status and cartesian data, output to other tasks
	m_masterStatus AT %Q* :ST_MasterStatus;
	
	// master robot joint data, output to other tasks
	m_masterJointsData AT %Q* :ST_MasterJointData;
		
	// master robot data, ouput to slave controller box
	m_masterRobotData AT %Q* :MSCommu_MasterStatus;
	
	// flag to init robot
	m_robotInit :BOOL :=FALSE;
	
	// wait time before robot init  for ethercat to be statble 
	m_robotInitWaitTime : LREAL:=0;
	
	// master robot
	m_masterRobot:FB_MasterRobot;
	
	// code execute time measure
	m_codeTime : Profiler;
	
END_VAR

m_codeTime(START:=TRUE, RESET:=TRUE);

// wait communication to be stable
IF(m_robotInitWaitTime<g_robotInitWaitTime) THEN
	m_robotInitWaitTime := m_robotInitWaitTime+g_armCtrlCycleTime;
	RETURN;
END_IF

// robot init
IF m_robotInit =FALSE THEN
	m_masterRobot.Init();
	m_robotInit:=TRUE;
END_IF

// input from UI
UIInputProcess();

// slave input data cast
slaveInputDataCast(m_slaveRobotData, m_masterInputDataPool.m_slaveStatus);

// robot run
m_masterRobot.run(m_masterInputDataPool);

// update data pool
m_masterRobot.getStatus(m_masterStatus,m_masterJointsData);

// master output data cast
masterOutputDataCast(m_masterRobot.m_shoulderPoseInMonitor, m_masterStatus, m_masterRobotData);

// output to UI
UIOutputProcess();

m_codeTime(START:=FALSE);

// convert from local ST_MasterStatus for control to MSCommu_MasterStatus for master-slave communication
METHOD masterOutputDataCast : BOOL
VAR_IN_OUT CONSTANT
	shoulderPose :ARRAY[1..2] OF ST_Frame;
	masterStatus :ST_MasterStatus;
END_VAR
VAR_IN_OUT
	masterOutputData:MSCommu_MasterStatus;
END_VAR

VAR
	i,j : INT;
	poseInMonitor:ST_Frame;
	velInShoulder, wVelInShoulder :Vec3d;
	velInMonitor, wVelInMonitor :Vec3d;
END_VAR
// Master heart beat
IF masterOutputData.m_heartBeat >= 10 THEN
	masterOutputData.m_heartBeat := 0;
ELSE
	masterOutputData.m_heartBeat := masterOutputData.m_heartBeat + 1;
END_IF

masterOutputData.m_motionScale :=masterStatus.m_motionScale;
masterOutputData.m_slaveSelfCheckFlag := m_masterInputDataPool.m_UIData.m_selfCheckFlag;
masterOutputData.m_pedalHover := m_masterInputDataPool.m_cartStatus.m_pedalHover;
masterOutputData.m_electricKnifePedalTrigger := m_masterInputDataPool.m_cartStatus.m_electricKnifePedalTrigger;
masterOutputData.m_tryMSControl[1] := BOOL_TO_INT(m_masterInputDataPool.m_cartStatus.m_surgonReady);
masterOutputData.m_tryMSControl[2] := BOOL_TO_INT(m_masterInputDataPool.m_cartStatus.m_surgonReady);
masterOutputData.m_uiResetFault := GVL_interactUI.g_uiResetFault;
masterOutputData.m_masterStopButton := NOT SafetyCheck.m_stopButton;

FOR i:=1 TO g_mArmNum DO
	masterOutputData.m_armState[i] := masterStatus.m_armState[i];
	masterOutputData.m_teleSlaveArmIdx[i] :=masterStatus.m_teleSlaveArmIdx[i];
	masterOutputData.m_gripAngle[i] := masterStatus.m_gripAngle[i] ;
	
	poseInMonitor := transform(shoulderPose[i],  masterStatus.m_curArmPose[i]);
	masterOutputData.m_curArmPose[i].m_pos := poseInMonitor.m_pos ;
	masterOutputData.m_curArmPose[i].m_rot := poseInMonitor.m_rot ;
	
	FOR j:=1 TO 3 DO
		velInShoulder[j]:=masterStatus.m_curArmTwist[i][j];
		wVelInShoulder[j]:=masterStatus.m_curArmTwist[i][j+3];
	END_FOR
	matMultiVec(shoulderPose[i].m_rot, velInShoulder,velInMonitor);
	matMultiVec(shoulderPose[i].m_rot, wVelInShoulder,wVelInMonitor);
	
	FOR j:=1 TO 3 DO
		masterOutputData.m_curArmTwist[i][j]:=velInMonitor[j];
		masterOutputData.m_curArmTwist[i][j+3]:=wVelInMonitor[j];
	END_FOR
END_FOR
END_METHOD

// convert from MSCommu_Slavetatus for master-slave communication to local ST_SlaveStatus for control
METHOD slaveInputDataCast : BOOL
VAR_IN_OUT CONSTANT
		slaveInputData : MSCommu_SlaveStatus; 
END_VAR
VAR_IN_OUT
	slaveStatus :ST_SlaveStatus;
END_VAR

VAR
	i :INT;
END_VAR
slaveStatus.m_selfCheckPass := slaveInputData.m_selfCheckPass;
slaveStatus.m_slaveHeartBeat := slaveInputData.m_heartBeat;
slaveStatus.m_endoscopeMounted :=slaveInputData.m_endoscopeMounted;
slaveStatus.m_endoscopePose.m_pos :=slaveInputData.m_endoscopePose.m_pos;
slaveStatus.m_endoscopePose.m_rot :=slaveInputData.m_endoscopePose.m_rot;
slaveStatus.m_asepticDeployCompleteFlag := slaveInputData.m_asepticDeployCompletedFlag;
slaveStatus.m_slaveStopButton := slaveInputData.m_slaveStopButton;
FOR i:= 1 TO g_sArmNum DO
	slaveStatus.m_armState[i] := slaveInputData.m_armState[i];
	slaveStatus.m_instruStauts[i].m_fingerAngle := slaveInputData.m_instruStauts[i].m_fingerAngle;
	slaveStatus.m_instruStauts[i].m_ready := slaveInputData.m_instruStauts[i].m_ready;
	slaveStatus.m_instruStauts[i].m_type := slaveInputData.m_instruStauts[i].m_type;
	slaveStatus.m_instruStauts[i].m_energyType := slaveInputData.m_instruEnergyType[i];
	slaveStatus.m_curArmPose[i].m_pos :=slaveInputData.m_curArmPose[i].m_pos;
	slaveStatus.m_curArmPose[i].m_rot :=slaveInputData.m_curArmPose[i].m_rot;
	slaveStatus.m_masterSlavePoseError[i] := slaveInputData.m_masterSlavePoseError[i];
END_FOR
END_METHOD

// tranform data from UI(global variable write by ADS) to ST_UIData
METHOD UIInputProcess : BOOL
VAR_INPUT
END_VAR
// master-slave control scale
IF 2 = GVL_interactUI.g_masterSlaveScaling THEN
	m_masterInputDataPool.m_UIData.m_motionScale := 2;
ELSIF 3 = GVL_interactUI.g_masterSlaveScaling THEN
	m_masterInputDataPool.m_UIData.m_motionScale := 3;
ELSE
	m_masterInputDataPool.m_UIData.m_motionScale := 1.5;
END_IF

// self-check
m_masterInputDataPool.m_UIData.m_selfCheckFlag := GVL_interactUI.g_slaveCheckEnbale;

// hand clutch
m_masterInputDataPool.m_UIData.m_enableHandClutch := GVL_interactUI.g_fingerClutchOnOff;

// arm disable
m_masterInputDataPool.m_UIData.m_masterArmDisableFlag[1]:=FALSE;
m_masterInputDataPool.m_UIData.m_masterArmDisableFlag[2]:=FALSE;
IF 1=GVL_interactUI.g_armIsDisbale OR 2=GVL_interactUI.g_armIsDisbale THEN
	m_masterInputDataPool.m_UIData.m_masterArmDisableFlag[GVL_interactUI.g_armIsDisbale] := TRUE;
END_IF
END_METHOD

METHOD UIOutputProcess : BOOL
VAR_INPUT
END_VAR
//slave arm self check status
IF m_masterInputDataPool.m_slaveStatus.m_armState[1] = SlaveArmState_SelfCheck OR m_masterInputDataPool.m_slaveStatus.m_armState[2] = SlaveArmState_SelfCheck OR 
			m_masterInputDataPool.m_slaveStatus.m_armState[3] = SlaveArmState_SelfCheck OR m_masterInputDataPool.m_slaveStatus.m_armState[4] = SlaveArmState_SelfCheck THEN
	GVL_interactUI.g_slaveCheckStatus := 1;
ELSIF m_masterInputDataPool.m_slaveStatus.m_selfCheckPass THEN
	GVL_interactUI.g_slaveCheckStatus := 2;
ELSE
	GVL_interactUI.g_slaveCheckStatus := 0;
END_IF

//GVL_interactUI.g_masterSelfCheckFinshed := m_masterStatus.m_selfCheckStatus;

GVL_interactUI.g_stateMachineArm1 := m_masterStatus.m_armState[1];
GVL_interactUI.g_stateMachineArm2 := m_masterStatus.m_armState[2];
GVL_interactUI.g_teleSlaveArm1Idx := m_masterStatus.m_teleSlaveArmIdx[1];
GVL_interactUI.g_teleSlaveArm2Idx := m_masterStatus.m_teleSlaveArmIdx[2];
GVL_interactUI.g_screenLockEnable := (MasterArmState_MasterSlave <= m_masterStatus.m_armState[1]  AND MasterArmState_Endoscope >= m_masterStatus.m_armState[1]) OR (MasterArmState_MasterSlave <= m_masterStatus.m_armState[2]  AND MasterArmState_Endoscope >= m_masterStatus.m_armState[2]);
IF m_masterInputDataPool.m_cartStatus.m_armSwitch THEN
	// ui reset variable
	GVL_interactUI.g_armSwitchEnable := 1;
END_IF
END_METHOD

END_PROGRAM

// ---- FBs_Robots/FB_MasterRobot.TcPOU
FUNCTION_BLOCK FB_MasterRobot
VAR
	// flag if slave are connected
	m_slaveOnLine :BOOL :=FALSE;
	m_slaveOnLineCheck :FB_slaveConnectionCheck;
	
	// master-slave motion scale
	m_motionScale :LREAL;
	
	// monitor angle
	m_monitorAngle :LREAL;
	
	// master arm base pose(shoulder pose) in monitor coordinate
	m_shoulderPoseInMonitor :ARRAY[1..2] OF ST_Frame;
	
	// master arms, responsible for arm kinematic and control
	m_masterArms :ARRAY[1..g_mArmNum] OF FB_MasterArm;
	
	// arm state
	m_masterArmState:ARRAY[1..g_mArmNum] OF E_masterArmState:=[E_masterArmState.MasterArmState_Init,E_masterArmState.MasterArmState_Error];
	m_lastMasterArmState:ARRAY[1..g_mArmNum] OF E_masterArmState:=[E_masterArmState.MasterArmState_Init,E_masterArmState.MasterArmState_Error];
	m_nextMasterArmState:ARRAY[1..g_mArmNum] OF E_masterArmState:=[E_masterArmState.MasterArmState_Init,E_masterArmState.MasterArmState_Error];
	
	// index(1 to 4) of slave arm which is tele-linked to master arm
	m_teleSlaveArmIdx:ARRAY[1..g_mArmNum] OF E_MatchedSlaveArmIdx:=[MatchedSlaveArmIdx_NULL, MatchedSlaveArmIdx_null];
	m_matchedMasterArmIdx :ST_MatchedMasterArmIdx;
	m_instruArmState:ARRAY [1..g_mArmNum] OF E_SlaveArmState:=[SlaveArmState_Error, SlaveArmState_Error];
	m_scopeArmState :E_SlaveArmState := SlaveArmState_Error;
	m_scopeArmIndex : E_MatchedSlaveArmIdx :=MatchedSlaveArmIdx_null;
	
	// flag if tele-manipulated slave arm is switched
	m_armSwitchFlag :ARRAY[1..2] OF BOOL := [2(FALSE)];
	
	//master arm selfcheck finshed flag
	m_armSelfCheckFinshedFlag :ARRAY [1..2] OF BOOL;
	
	// flag to enter master-slave control, triggerd by pinching the gripper twice in on second
	m_MSCtrlTriggerFlag :ARRAY[1..g_mArmNum] OF BOOL:=[FALSE, FALSE];
	m_MSCtrlTriggerCheck :ARRAY[1..g_mArmNum] OF FB_MSCtrlTriggerCheck;
	
	// all arm controller instance 
	m_armCtrlFactory :ARRAY[1..g_mArmNum,1..MasterArmState_totalNum] OF I_MasterArmCtrl;
	m_armError :ARRAY[1..g_mArmNum] OF FB_StateCtrlError;
	m_armInit :ARRAY[1..g_mArmNum] OF FB_StateCtrlInit;
	m_armHome :ARRAY[1..g_mArmNum] OF FB_StateCtrlHome;
	m_armStandBy :ARRAY[1..g_mArmNum] OF FB_StateCtrlStandBy;
	m_armMatching :ARRAY[1..g_mArmNum] OF FB_StateCtrlMatching;
	m_armReady :ARRAY[1..g_mArmNum] OF FB_StateCtrlReady;
	m_armMasterSlave :ARRAY[1..g_mArmNum] OF FB_StateCtrlMasterSlave;
	m_armClutch :ARRAY[1..g_mArmNum] OF FB_StateCtrlClutch;
	m_armEndoscope :ARRAY[1..g_mArmNum] OF FB_StateCtrlEndoscope;
	m_armCart :ARRAY[1..g_mArmNum] OF FB_StateCtrlCart;
	m_armGravityCali :ARRAY[1..g_mArmNum] OF FB_StateCtrlGraCali;
	m_armTest :ARRAY[1..g_mArmNum] OF FB_StateCtrlTest;
	m_armDisable :ARRAY[1..g_mArmNum] OF FB_StateCtrlDisable;
	m_armPerformance :ARRAY[1..g_mArmNum] OF FB_StateCtrlPerformance;
	m_armGravityBiasCali :ARRAY[1..g_mArmNum] OF FB_StateCtrlGraBiasCali;	
	
	// specialized endoscope controller
	m_scopeCtrl :FB_EndoscopeController;
	
	// arm controller interface
	m_armCtrl :ARRAY[1..g_mArmNum] OF I_MasterArmCtrl;
	m_armCtrlCmds :ARRAY[1..g_mArmNum] OF ST_ArmCtrlCmds;
	
	// ultrasonic knife rotation clutch flag
	m_USKnifeRotClutch :ARRAY[1..g_sArmNum] OF BOOL := [4(FALSE)];

END_VAR

 METHOD PROTECTED checkTeleSlaveArmIdx : BOOL
VAR_IN_OUT CONSTANT
	i_masterInputDataPool:ST_MasterInputDataPool;
END_VAR
VAR_STAT
	m_armSwitchR : R_TRIG;
	m_armSwitch : BOOL;
	nextTeleSlaveArmIdx:ARRAY[1..g_mArmNum] OF E_MatchedSlaveArmIdx;
END_VAR
nextTeleSlaveArmIdx:=m_teleSlaveArmIdx;
m_armSwitchR(CLK:= i_masterInputDataPool.m_cartStatus.m_armSwitch, Q=> m_armSwitch);
IF m_armSwitch THEN
	m_matchedMasterArmIdx.left1ArmIdx := GVL_interactUI.g_armDistributionInfo.m_leftMappingSlaveArm[1];
	m_matchedMasterArmIdx.left2ArmIdx := GVL_interactUI.g_armDistributionInfo.m_leftMappingSlaveArm[2];
	m_matchedMasterArmIdx.right1ArmIdx := GVL_interactUI.g_armDistributionInfo.m_rightMappingSlaveArm[1];
	m_matchedMasterArmIdx.right2ArmIdx := GVL_interactUI.g_armDistributionInfo.m_rightMappingSlaveArm[2];
END_IF


IF m_matchedMasterArmIdx.left1ArmIdx <=0 OR m_matchedMasterArmIdx.left2ArmIdx <=0 OR m_matchedMasterArmIdx.right1ArmIdx <=0 OR m_matchedMasterArmIdx.right2ArmIdx <=0 THEN
	RETURN;
END_IF

// switch tele-controlled arm index when arm is disenabled
IF i_masterInputDataPool.m_slaveStatus.m_armState[m_matchedMasterArmIdx.left1ArmIdx] = SlaveArmState_Disable THEN
	nextTeleSlaveArmIdx[1]:= m_matchedMasterArmIdx.left2ArmIdx;
ELSIF i_masterInputDataPool.m_slaveStatus.m_armState[m_matchedMasterArmIdx.left2ArmIdx] = SlaveArmState_Disable THEN
	nextTeleSlaveArmIdx[1]:= m_matchedMasterArmIdx.left1ArmIdx;
ELSIF i_masterInputDataPool.m_slaveStatus.m_armState[m_matchedMasterArmIdx.right1ArmIdx] = SlaveArmState_Disable THEN
	nextTeleSlaveArmIdx[2]:= m_matchedMasterArmIdx.right2ArmIdx;
ELSIF i_masterInputDataPool.m_slaveStatus.m_armState[m_matchedMasterArmIdx.right2ArmIdx] = SlaveArmState_Disable THEN
	nextTeleSlaveArmIdx[2]:= m_matchedMasterArmIdx.right1ArmIdx;
END_IF


// switch tele-controlled arm index when endoscope is mounted
IF m_scopeArmIndex = m_matchedMasterArmIdx.left1ArmIdx OR m_scopeArmIndex = m_matchedMasterArmIdx.left2ArmIdx THEN
	// left arm
	IF m_scopeArmIndex = m_matchedMasterArmIdx.left1ArmIdx THEN
		nextTeleSlaveArmIdx[1] := m_matchedMasterArmIdx.left2ArmIdx;
	ELSE
		nextTeleSlaveArmIdx[1] := m_matchedMasterArmIdx.left1ArmIdx;
	END_IF
	
	// right arm
	// switch tele-controlled arm index when arm switch is triggerd
	IF m_armSwitch THEN
		IF m_teleSlaveArmIdx[2] = m_matchedMasterArmIdx.right1ArmIdx AND i_masterInputDataPool.m_slaveStatus.m_armState[m_matchedMasterArmIdx.right2ArmIdx]=SlaveArmState_InstruReady THEN
			nextTeleSlaveArmIdx[2] := m_matchedMasterArmIdx.right2ArmIdx;
		ELSIF 
			m_teleSlaveArmIdx[2]=m_matchedMasterArmIdx.right2ArmIdx AND i_masterInputDataPool.m_slaveStatus.m_armState[m_matchedMasterArmIdx.right1ArmIdx]=SlaveArmState_InstruReady THEN
			nextTeleSlaveArmIdx[2] := m_matchedMasterArmIdx.right1ArmIdx;
		ELSE
			IF  i_masterInputDataPool.m_slaveStatus.m_armState[m_matchedMasterArmIdx.right1ArmIdx]=SlaveArmState_InstruReady THEN
				nextTeleSlaveArmIdx[2] := m_matchedMasterArmIdx.right1ArmIdx;
			ELSIF i_masterInputDataPool.m_slaveStatus.m_armState[m_matchedMasterArmIdx.right2ArmIdx]=SlaveArmState_InstruReady THEN
				nextTeleSlaveArmIdx[2] := m_matchedMasterArmIdx.right2ArmIdx;
			ELSE
				nextTeleSlaveArmIdx[2] := m_matchedMasterArmIdx.right1ArmIdx;
			END_IF
			
		END_IF
	END_IF

ELSIF m_scopeArmIndex = m_matchedMasterArmIdx.right1ArmIdx OR m_scopeArmIndex = m_matchedMasterArmIdx.right2ArmIdx THEN
	// left arm
	// switch tele-controlled arm index when arm switch is triggerd
	IF m_armSwitch THEN
		IF m_teleSlaveArmIdx[1]=m_matchedMasterArmIdx.left1ArmIdx AND i_masterInputDataPool.m_slaveStatus.m_armState[m_matchedMasterArmIdx.left2ArmIdx]=SlaveArmState_InstruReady THEN
			nextTeleSlaveArmIdx[1] := m_matchedMasterArmIdx.left2ArmIdx;
		ELSIF 
			m_teleSlaveArmIdx[1]=m_matchedMasterArmIdx.left2ArmIdx AND i_masterInputDataPool.m_slaveStatus.m_armState[m_matchedMasterArmIdx.left1ArmIdx]=SlaveArmState_InstruReady THEN
			nextTeleSlaveArmIdx[1] := m_matchedMasterArmIdx.left1ArmIdx;
		ELSE
			IF  i_masterInputDataPool.m_slaveStatus.m_armState[m_matchedMasterArmIdx.left1ArmIdx]=SlaveArmState_InstruReady THEN
				nextTeleSlaveArmIdx[1] := m_matchedMasterArmIdx.left1ArmIdx;
			ELSIF i_masterInputDataPool.m_slaveStatus.m_armState[m_matchedMasterArmIdx.left2ArmIdx]=SlaveArmState_InstruReady THEN
				nextTeleSlaveArmIdx[1] := m_matchedMasterArmIdx.left2ArmIdx;
			ELSE
				nextTeleSlaveArmIdx[1] := m_matchedMasterArmIdx.left1ArmIdx;
			END_IF
		END_IF
	END_IF

	// right arm
	IF m_scopeArmIndex = m_matchedMasterArmIdx.right1ArmIdx THEN
		nextTeleSlaveArmIdx[2] := m_matchedMasterArmIdx.right2ArmIdx;
	ELSE
		nextTeleSlaveArmIdx[2] := m_matchedMasterArmIdx.right1ArmIdx;
	END_IF
END_IF

// check if arm-switch is triggerd
m_armSwitchFlag[1]:=m_teleSlaveArmIdx[1] <>  nextTeleSlaveArmIdx[1];
m_armSwitchFlag[2]:=m_teleSlaveArmIdx[2] <>  nextTeleSlaveArmIdx[2];

m_teleSlaveArmIdx:= nextTeleSlaveArmIdx;
END_METHOD

METHOD PROTECTED controllerTransit : BOOL
VAR_INPUT
END_VAR
VAR
	i :INT;
END_VAR
FOR i:=1 TO g_mArmNum DO 
	IF m_nextMasterArmState[i]<> m_masterArmState[i] THEN
		// reset current controller
		m_armCtrl[i].reset();
		
		// transit to new controller
		m_lastMasterArmState[i]:=m_masterArmState[i];
		m_masterArmState[i]:=m_nextMasterArmState[i];
		m_armCtrl[i]:=m_armCtrlFactory[i,m_masterArmState[i]];
		
		// init next controller
		m_armCtrl[i].Init(m_masterArms[i],m_armCtrlCmds[i]);
		
		// init scope controller
		IF m_masterArmState[i] = MasterArmState_Endoscope  THEN
			m_scopeCtrl.init(m_shoulderPoseInMonitor, m_masterArms, m_armCtrlCmds);
		END_IF
		
		m_masterArms[i].updateCmds(m_armCtrlCmds[i]);
	END_IF
END_FOR
END_METHOD

METHOD PUBLIC getStatus : BOOL
VAR_IN_OUT
	// master robot information, including arm status and cartesian data
	r_masterStatus :ST_MasterStatus;
	
	// master robot joint data
	r_masterJointsData :ST_MasterJointData;
	
END_VAR

VAR
	i:INT;
END_VAR
r_masterStatus.m_motionScale := m_motionScale;
r_masterStatus.m_armState:=m_masterArmState;
r_masterStatus.m_teleSlaveArmIdx := m_teleSlaveArmIdx;
r_masterStatus.m_matchedMasterArmIdx := m_matchedMasterArmIdx;

FOR i:=1 TO g_mArmNum DO
	// current info
	r_masterStatus.m_gripAngle[i]:=m_masterArms[i].gripAngle;
	// cartesion
//	r_masterStatus.m_curArmPose[i]:=m_masterArms[i].curCartPose;
//	r_masterStatus.m_curArmTwist[i]:=m_masterArms[i].curCartTwist;
	r_masterStatus.m_curArmPose[i]:=m_masterArms[i].m_curCartLinkPose;
	r_masterStatus.m_curArmTwist[i]:=m_masterArms[i].m_curCartLinkTwist;
	// joint
	r_masterJointsData.m_curMotorPos[i]:=m_masterArms[i].curMotorPos;
	r_masterJointsData.m_curLinkPos[i]:=m_masterArms[i].curLinkPos;
	r_masterJointsData.m_curJntPos[i]:=m_masterArms[i].curJntPos;
	r_masterJointsData.m_curJntVel[i]:=m_masterArms[i].curJntVel;
	r_masterJointsData.m_curJntTrq[i]:=m_masterArms[i].curJntTrq;
	r_masterJointsData.m_rawJntCurrent[i]:=m_masterArms[i].rawJntCurrent;
	r_masterJointsData.m_filtJntCurrent[i]:=m_masterArms[i].filtJntCurrent;
	
	// command info
	// cartesion
	r_masterStatus.m_cmdArmPose[i]:=m_masterArms[i].m_cmdCartPose;
	r_masterStatus.m_cmdArmTwist[i]:=m_masterArms[i].m_cmdCartTwist;
	// joint info
	r_masterJointsData.m_cmdJntPos[i]:=m_masterArms[i].m_cmdJntPos;
	r_masterJointsData.m_cmdJntVel[i]:=m_masterArms[i].m_cmdJntVel;
	r_masterJointsData.m_cmdJntTrq[i]:=m_masterArms[i].m_cmdJntTrq;
	r_masterJointsData.m_cmdJntCurrent[i]:=m_masterArms[i].cmdJntCurrent;
	//data to safety check
	r_masterStatus.m_gripHallSensor[i] := m_masterArms[i].m_gripHallSensorIO;
	r_masterStatus.m_slaveOnLine := m_slaveOnLine;
	r_masterStatus.m_IKSuccess[i] := m_armMatching[i].IKSuccess;
	r_masterStatus.m_timePeriod[i] := m_armMatching[i].timePeriod;
	//r_masterStatus.m_selfCheckStatus
END_FOR
END_METHOD

METHOD PUBLIC Init : BOOL
VAR_INPUT
END_VAR
VAR
	i:INT;
END_VAR
// init tele-controlled arm index
m_teleSlaveArmIdx[1]:=MatchedSlaveArmIdx_1;
m_teleSlaveArmIdx[2]:=MatchedSlaveArmIdx_3;

// shoulder pose in monitor
m_shoulderPoseInMonitor[1].m_pos[1]:=-g_shoulderDistance/2;
m_shoulderPoseInMonitor[2].m_pos[1]:=g_shoulderDistance/2;

FOR i:=1 TO g_mArmNum DO
	// arm init
	m_masterArms[i].Init(i);
	m_masterArmState[i]:=MasterArmState_Init;
	m_lastMasterArmState[i]:=MasterArmState_Init;
	m_nextMasterArmState[i]:=MasterArmState_Init;
	
	// command init
	m_armCtrlCmds[i].m_jntEnableFlag := g_zeroVec7i;
	m_armCtrlCmds[i].m_jntOPMode := g_allPosMode;
	m_armCtrlCmds[i].m_cmdCartPose := m_masterArms[i].curCartPose;
	m_armCtrlCmds[i].m_cmdCartTwist := g_zeroVec6d;
	m_armCtrlCmds[i].m_cmdJntPos := m_masterArms[i].curJntPos;
	m_armCtrlCmds[i].m_cmdJntVel := g_zeroVec7d;
	m_armCtrlCmds[i].m_cmdJntAcc := g_zeroVec7d;
	m_armCtrlCmds[i].m_cmdJntTrq := g_zeroVec7d;
	
	// generate controller factory
	m_armCtrlFactory[i,MasterArmState_Error] := m_armError[i];
	m_armCtrlFactory[i,MasterArmState_Init] := m_armInit[i];
	m_armCtrlFactory[i,MasterArmState_Home] := m_armHome[i];
	m_armCtrlFactory[i,MasterArmState_Standby] := m_armStandBy[i];
	m_armCtrlFactory[i,MasterArmState_Matching] := m_armMatching[i];
	m_armCtrlFactory[i,MasterArmState_Ready] := m_armReady[i];
	m_armCtrlFactory[i,MasterArmState_MasterSlave] := m_armMasterSlave[i];
	m_armCtrlFactory[i,MasterArmState_Clutch] := m_armClutch[i];
	m_armCtrlFactory[i,MasterArmState_Endoscope] := m_armEndoscope[i];
	m_armCtrlFactory[i,MasterArmState_Cart] := m_armCart[i];
	m_armCtrlFactory[i,MasterArmState_GravityCali] := m_armGravityCali[i];
	m_armCtrlFactory[i,MasterArmState_Test] := m_armTest[i];
	m_armCtrlFactory[i,MasterArmState_Disable] := m_armDisable[i];
	m_armCtrlFactory[i,MasterArmState_Performance] := m_armPerformance[i];
	m_armCtrlFactory[i,MasterArmState_GravityBiasCali] := m_armGravityBiasCali[i];

	// assign controller
	m_armCtrl[i]:=m_armCtrlFactory[i,m_masterArmState[i]];
	m_armCtrl[i].Init(m_masterArms[i],m_armCtrlCmds[i]);
	
	// init master-slave trigger
	m_MSCtrlTriggerCheck[i].init(g_armCtrlCycleTime, 2);
END_FOR
END_METHOD

METHOD PROTECTED MSCtrlTriggerCheck : BOOL
VAR_IN_OUT CONSTANT
		i_masterInputDataPool:ST_MasterInputDataPool;
END_VAR
VAR
	i:INT;
END_VAR
FOR i:=1 TO g_mArmNum DO
	IF MasterArmState_Ready = m_masterArmState[i] AND SlaveArmState_InstruReady = m_instruArmState[i] 
		AND SlaveArmState_ScopeReady = m_scopeArmState AND i_masterInputDataPool.m_cartStatus.m_surgonReady THEN
		m_MSCtrlTriggerFlag[i]:=m_MSCtrlTriggerCheck[i].run(m_masterArms[i].gripAngle);
	END_IF
	
	IF  MatchedSlaveArmIdx_NULL =  m_teleSlaveArmIdx[i] OR   NOT(i_masterInputDataPool.m_cartStatus.m_surgonReady) 
		OR 	NOT(i_masterInputDataPool.m_slaveStatus.m_instruStauts[m_teleSlaveArmIdx[i]].m_ready) 
		OR m_masterArmState[i] = MasterArmState_Error OR i_masterInputDataPool.m_cartStatus.m_consoleInAdjust
		OR  SlaveArmState_Error = m_instruArmState[i] OR SlaveArmState_Disable = m_instruArmState[i]  THEN
		m_MSCtrlTriggerFlag[i]:=FALSE;
		m_MSCtrlTriggerCheck[i].reset();
	END_IF  
END_FOR
END_METHOD

METHOD PUBLIC run : BOOL
VAR_IN_OUT CONSTANT
	i_masterInputDataPool:ST_MasterInputDataPool;
END_VAR
VAR
	i:INT;
END_VAR
m_motionScale := i_masterInputDataPool.m_UIData.m_motionScale;
m_monitorAngle := i_masterInputDataPool.m_cartStatus.m_monitorAngle;

// check slave connection
m_slaveOnLine := m_slaveOnLineCheck.check(i_masterInputDataPool.m_slaveStatus.m_slaveHeartBeat);

// update shoulder pose
updateShoulderPose();

// check tele-operated slave arms index
checkTeleSlaveArmIdx(i_masterInputDataPool);

// check if to trig ultrasonic knife ratotation clutch
USKnifeClutchCheck(i_masterInputDataPool);

// update arm status
FOR i:=1 TO g_mArmNum DO
	// update dynamic data
	m_masterArms[i].updateDyna(i_masterInputDataPool.m_masterDynaData);
								
	// update master arm kinematics
	m_masterArms[i].updateStatus();
END_FOR

// state machine transition
stateMachine(i_masterInputDataPool);

// controller transition
controllerTransit();

// run arm controller
FOR i:=1 TO g_mArmNum DO
	// null ptr check
	ASSERT(0 <> m_armCtrl[i]);
	
	// run controller
	m_armCtrl[i].run(m_teleSlaveArmIdx[i], m_shoulderPoseInMonitor[i], m_masterArms[i],
						i_masterInputDataPool.m_slaveStatus,m_armCtrlCmds[i]);
						
	// update commands to drivers
	m_masterArms[i].updateCmds(m_armCtrlCmds[i]);
END_FOR

// run scope controller
IF m_masterArmState[1] = MasterArmState_Endoscope AND m_masterArmState[2] = MasterArmState_Endoscope THEN
	m_scopeCtrl.run(m_teleSlaveArmIdx, m_shoulderPoseInMonitor, m_masterArms, i_masterInputDataPool.m_slaveStatus, m_armCtrlCmds);
	m_masterArms[1].updateCmds(m_armCtrlCmds[1]);
	m_masterArms[2].updateCmds(m_armCtrlCmds[2]);
END_IF
END_METHOD

PROPERTY shoulderPose : ARRAY[1..2] OF ST_Frame
GET
shoulderPose := m_shoulderPoseInMonitor;
END_GET
END_PROPERTY

// state machine check and transit 
METHOD PROTECTED stateMachine : BOOL
VAR_IN_OUT CONSTANT
		i_masterInputDataPool:ST_MasterInputDataPool;
END_VAR
VAR
	i:INT;
	enableClutch :BOOL;
END_VAR
// get instrument arm state
FOR i:=1 TO g_mArmNum DO
	IF MatchedSlaveArmIdx_NULL =  m_teleSlaveArmIdx[i] THEN
		m_instruArmState[i] := SlaveArmState_Error;
	ELSE
		m_instruArmState[i] := i_masterInputDataPool.m_slaveStatus.m_armState[m_teleSlaveArmIdx[i]];
	END_IF
END_FOR

// get endoscope arm state
m_scopeArmState := SlaveArmState_Error;
m_scopeArmIndex := MatchedSlaveArmIdx_null;
FOR i:=1 TO g_sArmNum DO 
	IF InstruType_endoscope =  i_masterInputDataPool.m_slaveStatus.m_instruStauts[i].m_type THEN
		m_scopeArmState := i_masterInputDataPool.m_slaveStatus.m_armState[i];
		m_scopeArmIndex := i;
		EXIT;
	END_IF
END_FOR

// check if master-slave grip angle match
MSCtrlTriggerCheck(i_masterInputDataPool);

// State machine transit 
FOR i:=1 TO g_mArmNum DO
	
	// flag if enable clutch
	enableClutch :=  i_masterInputDataPool.m_cartStatus.m_clutchSwitch OR (m_masterArms[i].handClutchSwitch AND i_masterInputDataPool.m_UIData.m_enableHandClutch);
	
	CASE m_masterArmState[i] OF
		// error
		MasterArmState_Error:
			// to standby
			IF FALSE = i_masterInputDataPool.m_safetyData.m_masterErrFlag[i] THEN
				IF m_armSelfCheckFinshedFlag[i] THEN
					m_nextMasterArmState[i] := MasterArmState_Standby;
				ELSE
					m_nextMasterArmState[i]:=MasterArmState_Home;
				END_IF
			END_IF
			
		// init
		MasterArmState_Init:
			// to home
			IF m_armCtrl[i].isFinished THEN
				// NOTICE: multiple cycles joints back to center during initialization
				// 			need to reset joints encoder data again
				m_masterArms[i].initJntPos();
				m_armSelfCheckFinshedFlag[i] := FALSE;
				m_nextMasterArmState[i]:=MasterArmState_Home;
			END_IF

		//home
		MasterArmState_Home:
			IF m_armCtrl[i].isFinished  THEN
				m_armSelfCheckFinshedFlag[i] := TRUE;
				m_nextMasterArmState[i]:=MasterArmState_GravityBiasCali;
			END_IF
			
		//graivity bias calibration
		MasterArmState_GravityBiasCali:
			IF m_armCtrl[i].isFinished  THEN
				m_nextMasterArmState[i]:=MasterArmState_Standby;
				m_masterArms[i].jntGravityBias := m_armGravityBiasCali[i].m_gravityBias;
			END_IF
		
		//standby
		MasterArmState_Standby:
			// to matching
			IF SlaveArmState_InstruReady = m_instruArmState[i] AND SlaveArmState_ScopeReady = m_scopeArmState 
					AND i_masterInputDataPool.m_slaveStatus.m_asepticDeployCompleteFlag AND m_slaveOnLine THEN
				m_nextMasterArmState[i]:=MasterArmState_Matching;
			// to clutch
			ELSIF enableClutch THEN
				m_nextMasterArmState[i] := MasterArmState_Clutch; 
			// to cart
			ELSIF i_masterInputDataPool.m_cartStatus.m_monitorInAdjust THEN
				m_nextMasterArmState[i] := MasterArmState_Cart;
			END_IF
		
		//matching
		MasterArmState_Matching:
			// to ready
			IF m_armCtrl[i].isFinished THEN
				m_nextMasterArmState[i]:=MasterArmState_Ready;
			// to clutch
			ELSIF enableClutch THEN
				m_nextMasterArmState[i] := MasterArmState_Clutch; 
			// to standby
			ELSIF SlaveArmState_InstruReady <> m_instruArmState[i] OR SlaveArmState_ScopeReady <> m_scopeArmState
						OR m_armSwitchFlag[i] THEN
				m_nextMasterArmState[i]:=MasterArmState_Standby;
			// to cart
			ELSIF i_masterInputDataPool.m_cartStatus.m_monitorInAdjust THEN
				m_nextMasterArmState[i] := MasterArmState_Cart;
			END_IF
		
		//ready
		MasterArmState_Ready:
			// to standby
			IF SlaveArmState_InstruReady <> m_instruArmState[i] OR SlaveArmState_ScopeReady <> m_scopeArmState
					OR m_armSwitchFlag[i] THEN
				m_nextMasterArmState[i]:=MasterArmState_Standby;
			// to clutch
			ELSIF enableClutch THEN
				m_nextMasterArmState[i] := MasterArmState_Clutch; 
			// to cart
			ELSIF i_masterInputDataPool.m_cartStatus.m_monitorInAdjust THEN
				m_nextMasterArmState[i] := MasterArmState_Cart;
			// to master-slave
			ELSIF SlaveArmState_InstruReady = m_instruArmState[i] AND SlaveArmState_ScopeReady = m_scopeArmState 
					AND i_masterInputDataPool.m_cartStatus.m_surgonReady AND m_MSCtrlTriggerFlag[i] AND NOT(i_masterInputDataPool.m_cartStatus.m_consoleInAdjust) THEN
				m_nextMasterArmState[i] := MasterArmState_MasterSlave;
			ELSIF NOT i_masterInputDataPool.m_slaveStatus.m_asepticDeployCompleteFlag THEN
				m_nextMasterArmState[i]:=MasterArmState_Standby;
			END_IF
		
		//MasterSlave
		MasterArmState_MasterSlave:
			// to standdy
			IF  (SlaveArmState_InstruReady <> m_instruArmState[i] AND SlaveArmState_MasterSlave <> m_instruArmState[i])
				OR SlaveArmState_ScopeReady <> m_scopeArmState OR NOT(i_masterInputDataPool.m_cartStatus.m_surgonReady)
				OR m_armSwitchFlag[i] THEN
				m_nextMasterArmState[i]:=MasterArmState_Standby;
			// to clutch
			ELSIF enableClutch THEN
				m_nextMasterArmState[i] := MasterArmState_Clutch; 
			//to standby
			ELSIF NOT m_slaveOnLine THEN
				m_nextMasterArmState[i] := MasterArmState_Standby;
			END_IF
			
		//Clutch
		MasterArmState_Clutch:
			// to standby
			IF NOT(enableClutch) THEN
				m_nextMasterArmState[i]:=MasterArmState_Standby;
			END_IF
		
		// Endoscope 
		MasterArmState_Endoscope:
			// to standby
			IF NOT(i_masterInputDataPool.m_cartStatus.m_surgonReady) OR NOT(i_masterInputDataPool.m_cartStatus.m_endoscopeSwitch) 
				OR (SlaveArmState_ScopeReady <> m_scopeArmState AND SlaveArmState_EndoScope <> m_scopeArmState) THEN
				m_nextMasterArmState[i] := MasterArmState_Standby;
			// to clutch
			ELSIF enableClutch THEN
				m_nextMasterArmState[i] := MasterArmState_Clutch; 
			//to standby
			ELSIF NOT m_slaveOnLine THEN
				m_nextMasterArmState[i] := MasterArmState_Standby;
			END_IF
			
		// Cart 
		MasterArmState_Cart:
			// to standby
			IF NOT( i_masterInputDataPool.m_cartStatus.m_consoleInAdjust) THEN
				m_nextMasterArmState[i] := MasterArmState_Standby;
			END_IF
		
		//Gravity Calibration
		MasterArmState_GravityCali:
			// to standby
			IF  m_armCtrl[i].isFinished THEN
				m_nextMasterArmState[i]:=MasterArmState_Standby;
			END_IF
	
		//arm test
		MasterArmState_Test:
			// to standby
			IF  m_armCtrl[i].isFinished THEN
				m_nextMasterArmState[i]:=MasterArmState_Standby;
			END_IF
			
		//arm Performance
		MasterArmState_Performance:
			// to standby
			IF  m_armCtrl[i].isFinished THEN
				m_nextMasterArmState[i]:=MasterArmState_Standby;
			END_IF
			
		//arm disable
		MasterArmState_Disable:
			// to init
			IF  NOT(i_masterInputDataPool.m_UIData.m_masterArmDisableFlag[i]) THEN
				m_armSelfCheckFinshedFlag[i] := FALSE;
				m_nextMasterArmState[i]:=MasterArmState_Init;
			END_IF
	END_CASE
	
	// arm disable
	IF i_masterInputDataPool.m_UIData.m_masterArmDisableFlag[i] THEN
		m_nextMasterArmState[i] := MasterArmState_Disable;
	// error check
	ELSIF i_masterInputDataPool.m_safetyData.m_masterErrFlag[i] THEN
		m_nextMasterArmState[i] := MasterArmState_Error;
	END_IF
	
END_FOR

// To Endoscope Control 
IF SlaveArmState_ScopeReady = m_scopeArmState AND i_masterInputDataPool.m_cartStatus.m_endoscopeSwitch AND i_masterInputDataPool.m_cartStatus.m_surgonReady AND
  (MasterArmState_Standby = m_masterArmState[1] OR MasterArmState_Ready = m_masterArmState[1] OR MasterArmState_Matching = m_masterArmState[1] OR MasterArmState_MasterSlave = m_masterArmState[1]) AND 
  (MasterArmState_Standby = m_masterArmState[2] OR MasterArmState_Ready = m_masterArmState[2] OR MasterArmState_Matching = m_masterArmState[2] OR MasterArmState_MasterSlave = m_masterArmState[2]) THEN
	m_nextMasterArmState[1] := MasterArmState_Endoscope;
	m_nextMasterArmState[2] := MasterArmState_Endoscope;
END_IF
END_METHOD

METHOD PROTECTED updateShoulderPose : BOOL
VAR_INPUT
END_VAR
VAR
	monitorRot :mat3d;
END_VAR
// base monitor frame(0 rotation angle) in current monitor frame 
monitorRot := rotY( -m_monitorAngle);

// shoulder pose in current monitor frame
matMultiply(g_shoulderRotInMonitor,monitorRot, m_shoulderPoseInMonitor[1].m_rot);
m_shoulderPoseInMonitor[2].m_rot:=m_shoulderPoseInMonitor[1].m_rot;
END_METHOD

METHOD USKnifeClutchCheck : BOOL
VAR_IN_OUT CONSTANT
	i_masterInputDataPool:ST_MasterInputDataPool;
END_VAR

VAR
	i:INT;
END_VAR
FOR i:=1 TO g_sArmNum DO
	IF NOT(i_masterInputDataPool.m_slaveStatus.m_instruStauts[i].m_ready) THEN
		m_USKnifeRotClutch[i] := FALSE;
	END_IF
END_FOR

FOR i:=1 TO g_mArmNum DO
	IF (i_masterInputDataPool.m_slaveStatus.m_instruStauts[m_teleSlaveArmIdx[i]].m_type = InstruType_UltrasoundKnifeS OR i_masterInputDataPool.m_slaveStatus.m_instruStauts[m_teleSlaveArmIdx[i]].m_type = InstruType_UltrasoundKnifeU)
		AND  m_masterArmState[i] = MasterArmState_Clutch AND m_masterArms[i].handClutchSwitch THEN
		m_USKnifeRotClutch[m_teleSlaveArmIdx[i]] := TRUE;
	END_IF
END_FOR
END_METHOD

END_FUNCTION_BLOCK

// ---- FBs_StateControllers/FB_StateCtrlError.TcPOU
// Brief: Master Arm Error Hold
FUNCTION_BLOCK PUBLIC FB_StateCtrlError EXTENDS FB_MasterArmCtrlBase
VAR_INPUT
END_VAR
VAR_OUTPUT
END_VAR
VAR
END_VAR

// override this function in each exact controller
METHOD PROTECTED calcCmdJntPos : BOOL
VAR_IN_OUT CONSTANT
	i_slaveIdx :INT;
	i_shoulderPose :ST_Frame;
	i_masterArm :FB_MasterArm;
	i_slaveStatus :ST_SlaveStatus;
END_VAR

VAR
	i:int;
END_VAR
FOR i := 1 TO g_mJntNum DO
	IF  m_jntEnableFlag[i] = 0 THEN
		m_cmdJntPos[i]:=i_masterArm.curJntPos[i];
	END_IF
END_FOR
END_METHOD

METHOD PUBLIC init : BOOL
VAR_IN_OUT CONSTANT
	i_masterArm	:FB_MasterArm;
END_VAR
VAR_IN_OUT 
	r_masterArmCtrlCmd :ST_ArmCtrlCmds;
END_VAR

VAR
	i:INT;
END_VAR
SUPER^.Init(i_masterArm,r_masterArmCtrlCmd);

//disable joints which is error
FOR i := 1 TO g_mJntNum DO
	IF SafetyCheck.m_SafetyCheck.m_jntErrFlag[i_masterArm.armIdx, i, 2] OR SafetyCheck.m_SafetyCheck.m_jntErrFlag[i_masterArm.armIdx, i, 3] THEN
		m_jntEnableFlag[i] := 0;
	ELSE
		m_jntEnableFlag[i] := 1;
	END_IF
END_FOR

// update commands to arm
copyCmds(r_masterArmCtrlCmd);
END_METHOD

END_FUNCTION_BLOCK

// ---- FBs_StateControllers/FB_MasterArmCtrlBase.TcPOU
// Master Arm Base Controller, Hold at Current Posture
FUNCTION_BLOCK FB_MasterArmCtrlBase IMPLEMENTS I_MasterArmCtrl
VAR_INPUT
END_VAR
VAR_OUTPUT
END_VAR
VAR
	// flag if the controller has finished all its jobs
	m_isFinished:BOOL:=FALSE;
	
	// controller execute time period
	m_timePeriod :LREAL:=0;
	
	// flag to hold last commands
	m_holdLastCmds :BOOL := FALSE;
	
	// arm control data
	m_cmdJntPos : VEC7d;
	m_cmdJntVel : VEC7d;
	m_cmdJntAcc : VEC7d;
	m_cmdJntTrq : VEC7d;
	m_jntOPMode : Vec7i;
	m_jntEnableFlag :Vec7i;
	m_cmdCartPose : ST_Frame;
	m_cmdCartTwist : Vec6d;
END_VAR

// override this function in each exact controller
METHOD PROTECTED calcCmdJntPos : BOOL

VAR_IN_OUT CONSTANT
	i_slaveIdx :INT;
	i_shoulderPose :ST_Frame;
	i_masterArm :FB_MasterArm;
	i_slaveStatus :ST_SlaveStatus;
END_VAR
END_METHOD

// override this function in each exact controller
METHOD PROTECTED calcCmdJntTrq : BOOL

VAR_IN_OUT CONSTANT
	i_slaveIdx :INT;
	i_shoulderPose :ST_Frame;
	i_masterArm :FB_MasterArm;
	i_slaveStatus :ST_SlaveStatus;
END_VAR
// set joint torque to zero in default
m_cmdJntTrq := g_zeroVec7d;
END_METHOD

METHOD checkToHoldLastCmds : BOOL
VAR_IN_OUT CONSTANT
	i_masterArm :FB_MasterArm;
END_VAR
VAR
	j:INT;
	maxJntErr:LREAL;
	jntCtrlErr:Vec7d;
END_VAR
// check if to hold the command joint position unchanged
vecSub(i_masterArm.m_cmdJntPos, i_masterArm.m_curJntPos,jntCtrlErr);
maxJntErr:=0.0;
FOR j:=1 TO g_mJntNum DO
	maxJntErr:= MAX(maxJntErr, ABS(jntCtrlErr[j]));
END_FOR

checkToHoldLastCmds := (maxJntErr<g_jntCtrlErrForCmdHold);
END_METHOD

METHOD copyCmds : BOOL
VAR_IN_OUT 
	r_masterArmCtrlCmd :ST_ArmCtrlCmds;
END_VAR
r_masterArmCtrlCmd.m_jntEnableFlag :=m_jntEnableFlag;
r_masterArmCtrlCmd.m_cmdCartPose:=m_cmdCartPose;
r_masterArmCtrlCmd.m_cmdCartTwist:=m_cmdCartTwist;
r_masterArmCtrlCmd.m_cmdJntPos:=m_cmdJntPos;
r_masterArmCtrlCmd.m_cmdJntVel:=m_cmdJntVel;
r_masterArmCtrlCmd.m_cmdJntAcc:=m_cmdJntAcc;
r_masterArmCtrlCmd.m_cmdJntTrq:=m_cmdJntTrq;
r_masterArmCtrlCmd.m_jntOPMode:=m_jntOPMode;
END_METHOD

// override this function in each exact controller
// NOTICE: set joint control mode here, and do some initialization if needed
METHOD PUBLIC init : BOOL
VAR_IN_OUT CONSTANT
	i_masterArm	:FB_MasterArm;
END_VAR
VAR_IN_OUT 
	r_masterArmCtrlCmd :ST_ArmCtrlCmds;
END_VAR
m_timePeriod:=0;
m_jntEnableFlag :=g_onesVec7i;
m_jntOPMode:=g_allPosTrqMode;
m_cmdCartPose:=i_masterArm.curCartPose;
m_cmdCartTwist:=g_zeroVec6d;
IF FALSE = m_holdLastCmds THEN
	m_cmdJntPos:=i_masterArm.curJntPos;
ELSE 
	m_cmdJntPos := r_masterArmCtrlCmd.m_cmdJntPos;
END_IF
m_cmdJntVel:=g_zeroVec7d;
m_cmdJntAcc:=g_zeroVec7d;
m_cmdJntTrq:=g_zeroVec7d;

// update commands to arm
copyCmds(r_masterArmCtrlCmd);
END_METHOD

PROPERTY isFinished : BOOL
GET
isFinished:=m_isFinished;
END_GET
END_PROPERTY

{warning '添加方法实现'}
METHOD reset : BOOL
m_isFinished:=FALSE;
END_METHOD

{warning '添加方法实现'}
METHOD run : BOOL

VAR_IN_OUT CONSTANT
	i_slaveIdx :INT;
	i_shoulderPose :ST_Frame;
	i_masterArm :FB_MasterArm;
	i_slaveStatus :ST_SlaveStatus;
END_VAR
VAR_IN_OUT
	r_masterArmCtrlCmd :ST_ArmCtrlCmds;
END_VAR
VAR
	i:INT;
END_VAR
IF m_isFinished THEN
	RETURN;
END_IF

// check if arm enabled
IF FALSE = i_masterArm.isEnabled(m_jntEnableFlag) THEN
	RETURN;
END_IF

// calculate command joint position--Motion control
calcCmdJntPos(i_slaveIdx, i_shoulderPose, i_masterArm,i_slaveStatus);

// calculate command joint torque -- Force control
calcCmdJntTrq(i_slaveIdx, i_shoulderPose, i_masterArm,i_slaveStatus);

// update commands to arm
copyCmds(r_masterArmCtrlCmd);

// update time period
m_timePeriod := m_timePeriod+g_armCtrlCycleTime;
END_METHOD

PROPERTY timePeriod : Lreal
GET
timePeriod := m_timePeriod;
END_GET
END_PROPERTY

END_FUNCTION_BLOCK

// ---- FBs_StateControllers/FB_StateCtrlInit.TcPOU
// Brief: Master Arm Master Slave Control
FUNCTION_BLOCK PUBLIC FB_StateCtrlInit EXTENDS FB_MasterArmCtrlBase
VAR_INPUT
END_VAR
VAR_OUTPUT
END_VAR
VAR
	m_jnt7SelfCheckVel : LREAL :=180*g_deg2Rad;
	m_jnt7HalfMotionRange : LREAL := 1.75*PI+0.26;
	m_jnt7LimitErr :LREAL := 5*g_deg2Rad;
	m_jnt7CenterPos :LREAL;
	// 0: driver on; 1: joint 7 move to upper limit, 2: joint 7 mvoe to center
	m_initState :INT :=0;
END_VAR

// override this function in each exact controller
METHOD PROTECTED calcCmdJntPos : BOOL

VAR_IN_OUT CONSTANT
	i_slaveIdx :INT;
	i_shoulderPose :ST_Frame;
	i_masterArm :FB_MasterArm;
	i_slaveStatus :ST_SlaveStatus;
END_VAR

VAR
	centerVel:LREAL;
//	curJntPos:Vec7d;
END_VAR
IF m_isFinished THEN
	RETURN;
END_IF

IF m_timePeriod > 1 THEN
	m_isFinished :=true;
END_IF
//CASE m_initState OF
//	0:
//		m_cmdJntPos := i_masterArm.curJntPos;
//		IF i_masterArm.isEnabled(m_jntEnableFlag) = TRUE THEN
//			m_initState :=1;
//		END_IF
//	1: 
//		m_cmdJntPos[7] := m_cmdJntPos[7] + m_jnt7SelfCheckVel * g_armCtrlCycleTime;
//		IF m_cmdJntPos[7]-i_masterArm.curJntPos[7] > m_jnt7LimitErr THEN
//			m_cmdJntPos[7]:=i_masterArm.curJntPos[7];
//			m_jnt7CenterPos :=m_cmdJntPos[7]-m_jnt7HalfMotionRange;
//			m_initState :=2;
//		END_IF
//	2:
//		centerVel :=LIMIT(-m_jnt7SelfCheckVel,(m_jnt7CenterPos-m_cmdJntPos[7])/g_armCtrlCycleTime,m_jnt7SelfCheckVel);
//		m_cmdJntPos[7] := m_cmdJntPos[7] + centerVel * g_armCtrlCycleTime;
//		IF ABS(m_jnt7CenterPos-i_masterArm.curJntPos[7]) < g_jntCtrlAngTolLow THEN
//			m_isFinished :=TRUE;
//		END_IF
//END_CASE
END_METHOD

METHOD PUBLIC init : BOOL
VAR_IN_OUT CONSTANT
	i_masterArm	:FB_MasterArm;
END_VAR
VAR_IN_OUT 
	r_masterArmCtrlCmd :ST_ArmCtrlCmds;
END_VAR

VAR
	i:INT;
END_VAR
SUPER^.Init(i_masterArm,r_masterArmCtrlCmd);
m_jntOPMode:=g_allPosMode;
m_initState :=0;

m_jntOPMode := g_allPosTrqMode;
END_METHOD

END_FUNCTION_BLOCK

// ---- FBs_StateControllers/FB_StateCtrlHome.TcPOU
// Brief: Master Arm Home Posture
FUNCTION_BLOCK PUBLIC FB_StateCtrlHome EXTENDS FB_MasterArmCtrlBase
VAR_INPUT
END_VAR
VAR_OUTPUT
END_VAR
VAR
	m_homePlanner : FB_TrajMoveJ;
	
END_VAR

// override this function in each exact controller
METHOD PROTECTED calcCmdJntPos : BOOL
VAR_IN_OUT CONSTANT
	i_slaveIdx :INT;
	i_shoulderPose :ST_Frame;
	i_masterArm :FB_MasterArm;
	i_slaveStatus :ST_SlaveStatus;
END_VAR
VAR 
	i :INT;
	curJntVel :Vec7d;
END_VAR
// check if planner is ready
IF m_homePlanner.isGene = FALSE THEN
	calcCmdJntPos:=FALSE;
	RETURN;
END_IF

// traj plan
calcCmdJntPos :=m_homePlanner.evaluate(m_timePeriod, jntPos=> m_cmdJntPos, jntVel=>m_cmdJntVel, jntAcc=> m_cmdJntAcc);

// check if to terminate
curJntVel :=i_masterArm.curJntVel;
m_isFinished :=m_timePeriod > m_homePlanner.duration  AND norm(curJntVel)<7*g_jntStaticVelThres;
END_METHOD

METHOD PUBLIC init : BOOL
VAR_IN_OUT CONSTANT
	i_masterArm	:FB_MasterArm;
END_VAR
VAR_IN_OUT 
	r_masterArmCtrlCmd :ST_ArmCtrlCmds;
END_VAR

VAR
	i,j :INT;
	startJntPos,endJntPos :Vec7d;
END_VAR
SUPER^.Init(i_masterArm,r_masterArmCtrlCmd);

// traj plan
startJntPos:=i_masterArm.curJntPos;
FOR j:=1 TO 7 DO 
endJntPos[j]:=g_homePosture[i_masterArm.armIdx,j];
END_FOR
m_homePlanner.init(startJntPos,endJntPos,g_homeMaxjntVel,g_homeMaxjntAcc,g_homeMaxjntJerk);

// update commands to arm
copyCmds(r_masterArmCtrlCmd);
END_METHOD

END_FUNCTION_BLOCK

// ---- FBs_StateControllers/FB_StateCtrlMatching.TcPOU
// Brief: Master Arm Orientation Matching
FUNCTION_BLOCK PUBLIC FB_StateCtrlMatching EXTENDS FB_MasterArmCtrlBase
VAR_INPUT
END_VAR
VAR_OUTPUT
END_VAR
VAR
	// master-slave orientation match threshold
	m_matchAngleThres :LREAL := 2*g_deg2Rad;
	
	m_cmdRotInMonitor :Mat3d;
	
	m_initSolvedJntPos, m_iteSovlvedJntPos :Vec7d;
	m_IKSuccess :BOOL;
	
	m_matchTrajPlanner : FB_TrajMoveJ;
	m_targetJntPos :Vec7d;
	
	m_maxMatchJntVel:Vec7d:=[1.0, 1.0, 1.0, 2*pi, 3*pi, 3*pi, 5*pi];
	m_maxMatchJntAcc:Vec7d:=[1.0, 1.0, 1.0,  8*pi, 12*pi, 12*pi, 20*pi];
	m_maxMatchJntJerk:Vec7d:=[7(100.0)];
	
	m_rotErrAng :LREAL;

END_VAR

// override this function in each exact controller
METHOD PROTECTED calcCmdJntPos : BOOL

VAR_IN_OUT CONSTANT
	i_slaveIdx :INT;
	i_shoulderPose :ST_Frame;
	i_masterArm :FB_MasterArm;
	i_slaveStatus :ST_SlaveStatus;
END_VAR
var 
	i,j : INT;

	mq4,mq5,mq6,mq7:LREAL;
	q4,q5,q6,q7:LREAL;

	rotErr:Mat3d;
	wristRotInJnt3, wristRotInJnt4 :Mat3d;
	rot, invRot :Mat3d;
	cycleNum:INT;
	
	jnt4MoveRange:LREAL;
	jnt5Bias, jnt4MoveScale :LREAL;
	
	curJntPos, curJntErr:Vec7d;

END_VAR
IF m_IKSuccess THEN 
	// check if planner is ready
	IF  m_matchTrajPlanner.isGene = FALSE THEN
		RETURN;
	END_IF
	
	// traj plan
	calcCmdJntPos :=m_matchTrajPlanner.evaluate(m_timePeriod, jntPos=> m_cmdJntPos, jntVel=>m_cmdJntVel, jntAcc=> m_cmdJntAcc);
	curJntPos :=i_masterArm.curJntPos;
	vecSub(m_targetJntPos, curJntPos, curJntErr);
	
	matTranspose(i_masterArm.curCartPose.m_rot, invRot);
	matMultiply(invRot, m_cmdCartPose.m_rot, rotErr);
	rot2AngAxis(rotErr, angle=>m_rotErrAng,axis=>);
	m_isFinished := m_timePeriod > m_matchTrajPlanner.duration AND  norm(curJntErr)<g_jntCtrlAngTolHigh;
	
	RETURN;
END_IF

// command rotation in monitor
m_cmdRotInMonitor := i_slaveStatus.m_curArmPose[i_slaveIdx].m_rot;

// command rotation in master arm base
matTranspose(i_shoulderPose.m_rot, invRot);
matMultiply(invRot, m_cmdRotInMonitor, m_cmdCartPose.m_rot);
m_cmdCartPose.m_pos:= i_masterArm.curCartPose.m_pos;

// calculate current orientation error
matTranspose(i_masterArm.curCartPose.m_rot, invRot);
matMultiply(invRot, m_cmdCartPose.m_rot, rotErr);
rot2AngAxis(rotErr, angle=>m_rotErrAng,axis=>);

// try IK with optimized posture
rot:=calcJnt3Rotation(m_cmdJntPos[1],m_cmdJntPos[2],m_cmdJntPos[3]);
matTranspose(rot, invRot);
matMultiply(invRot, m_cmdCartPose.m_rot, wristRotInJnt3);
IF 1=i_masterArm.armIdx THEN
	m_IKSuccess := leftWristOptIK(wristRotInJnt3,q4=>q4, q5=>q5, q6=>q6, q7=>q7);
ELSE
	m_IKSuccess := rightWristOptIK(wristRotInJnt3,q4=>q4, q5=>q5, q6=>q6, q7=>q7);
END_IF

// try IK with joint4 at minimal limit
IF NOT m_IKSuccess THEN
	q4:= GVL_ArmJointParameters.g_minJntPos[i_masterArm.armIdx,4];
	
	rot:=calcJnt4Rotation(m_cmdJntPos[1],m_cmdJntPos[2],m_cmdJntPos[3],q4);
	matTranspose(rot, invRot);
	matMultiply(invRot, m_cmdCartPose.m_rot, wristRotInJnt4);
	m_IKSuccess := wristIK(wristRotInJnt4,i_masterArm, q5=>q5, q6=>q6, q7=>q7);
END_IF

// try IK with joint4 at maximum limit
IF NOT m_IKSuccess THEN
	q4:= GVL_ArmJointParameters.g_maxJntPos[i_masterArm.armIdx,4];
	
	rot:=calcJnt4Rotation(m_cmdJntPos[1],m_cmdJntPos[2],m_cmdJntPos[3],q4);
	matTranspose(rot, invRot);
	matMultiply(invRot, m_cmdCartPose.m_rot, wristRotInJnt4);
	m_IKSuccess := wristIK(wristRotInJnt4,i_masterArm, q5=>q5, q6=>q6, q7=>q7);
END_IF

// minimize joint4 move angle
IF m_IKSuccess THEN
	
	// minimize based on join5 posture
	jnt4MoveRange :=  i_masterArm.jnt4LinkToMotor(m_targetJntPos[2],m_targetJntPos[3],q4)-i_masterArm.curJntPos[4];
	jnt5Bias :=  LIMIT (0, ABS(q5-pi), pi/2);
	jnt4MoveRange := jnt4MoveRange * ABS(COS(jnt5Bias));
	
	// minimize based on cartesian error
	IF ABS(m_rotErrAng)< 5.0 * g_deg2Rad THEN
		jnt4MoveRange := 0.0;
	END_IF
	
	mq4:=  i_masterArm.jnt4MotorToLink(m_targetJntPos[2],m_targetJntPos[3],i_masterArm.curJntPos[4] + jnt4MoveRange) ;
	
	rot:=calcJnt4Rotation(m_cmdJntPos[1],m_cmdJntPos[2],m_cmdJntPos[3],mq4);
	matTranspose(rot, invRot);
	matMultiply(invRot, m_cmdCartPose.m_rot, wristRotInJnt4);
	IF wristIK(wristRotInJnt4,i_masterArm, q5=>mq5, q6=>mq6, q7=>mq7) THEN
		q4:=mq4;
		q5:=mq5;
		q6:=mq6;
		q7:=mq7;
	END_IF
END_IF

// traj plan
IF m_IKSuccess THEN 
	m_targetJntPos:=m_cmdJntPos;
	m_targetJntPos[4]:=i_masterArm.jnt4LinkToMotor(m_targetJntPos[2],m_targetJntPos[3],q4);
	m_targetJntPos[5]:=q5;
	m_targetJntPos[6]:=q6;
	
	// roll flip handle
	i_masterArm.flipGripper(rollFlipHandle(i_masterArm.armIdx,i_masterArm.curJntPos[7], q7, o_cmdJntPos7 =>m_targetJntPos[7]));
	
	// no match for rotate joint if instrument is ultrasonic knife
	IF MasterArmControl.m_masterRobot.m_USKnifeRotClutch[i_slaveIdx] THEN
		m_targetJntPos[7] := i_masterArm.curJntPos[7];
	END_IF

	m_matchTrajPlanner.init(m_cmdJntPos,m_targetJntPos,m_maxMatchJntVel,m_maxMatchJntAcc,m_maxMatchJntJerk);
	m_timePeriod :=0;
END_IF
END_METHOD

// calculate joint3 rotation in arm coordinate
(*armDH=[   0      0   q1      d1;
            -deg90  0   q2      0;
            0       a3  q3      0];*)
METHOD PROTECTED calcJnt3Rotation : Mat3d
VAR_INPUT CONSTANT
	q1:LREAL;
	q2:LREAL;
	q3:LREAL;
END_VAR

VAR
	c1,c2,c3,s1,s2,s3,c23,s23 :LREAL;
END_VAR
// !Convert active joint position to DH model for kinematic calculation
q3:=q3-q2;  //q3=q8-q2

c1:=COS(q1);
c2:=COS(q2);
c3:=COS(q3);

s1:=SIN(q1);
s2:=SIN(q2);
s3:=SIN(q3);

c23:=COS(q2+q3);
s23:=SIN(q2+q3);

calcJnt3Rotation[1,1]:= c23*c1;
calcJnt3Rotation[2,1]:= c23*s1;
calcJnt3Rotation[3,1]:= -s23;

calcJnt3Rotation[1,2]:= -s23*c1;
calcJnt3Rotation[2,2]:= -s23*s1;
calcJnt3Rotation[3,2]:= -c23;

calcJnt3Rotation[1,3]:= -s1;
calcJnt3Rotation[2,3]:= c1;
calcJnt3Rotation[3,3]:=0;
END_METHOD

// calculate joint3 rotation in arm coordinate
(*[   0      0   q1      d1;
	-deg90  0   q2      0;
	0       a3  q3      0;
	 -deg90  a4  q4      d4]
*)
METHOD PROTECTED calcJnt4Rotation : Mat3d
VAR_INPUT
	q1 :LREAL;
	q2 :LREAL;
	q3 :LREAL;
	q4 :LREAL;// already at the link side
END_VAR

VAR
	c1,c2,c3,c4, s1,s2,s3,s4,c23,s23 :LREAL;
END_VAR
// !Convert active joint position to DH model for kinematic calculation
//q4:=q4+q3-q2-pi/2;//q4DH=q4motor+q8-q2-90;  
q3:=q3-q2;  //q3=q8-q2

c1:=COS(q1);
c2:=COS(q2);
c3:=COS(q3);
c4:=COS(q4);

s1:=SIN(q1);
s2:=SIN(q2);
s3:=SIN(q3);
s4:=SIN(q4);

c23:=COS(q2+q3);
s23:=SIN(q2+q3);

calcJnt4Rotation[1,1]:= s1*s4 + c4*c1*c23;
calcJnt4Rotation[2,1]:= - c1*s4 + c4*s1*c23;
calcJnt4Rotation[3,1]:= -s23*c4;

calcJnt4Rotation[1,2]:= c4*s1 - s4*c1*c23;
calcJnt4Rotation[2,2]:= -s4*s1*c23 - c1*c4;
calcJnt4Rotation[3,2]:=   s23*s4;

calcJnt4Rotation[1,3]:= -s23*c1;
calcJnt4Rotation[2,3]:= -s23*s1;
calcJnt4Rotation[3,3]:=-c23;
END_METHOD

PROPERTY IKSuccess : BOOL
GET
IKSuccess := m_IKSuccess;
END_GET
END_PROPERTY

METHOD PUBLIC init : BOOL
VAR_IN_OUT CONSTANT
	i_masterArm	:FB_MasterArm;
END_VAR
VAR_IN_OUT 
	r_masterArmCtrlCmd :ST_ArmCtrlCmds;
END_VAR
// check if to hold the command joint position unchanged
m_holdLastCmds := checkToHoldLastCmds(i_masterArm);

// init
SUPER^.Init(i_masterArm,r_masterArmCtrlCmd);

m_jntOPMode[4]:=DriverOPMode_PosTrq;
m_jntOPMode[5]:=DriverOPMode_PosTrq;
m_jntOPMode[6]:=DriverOPMode_PosTrq;
m_jntOPMode[7]:=DriverOPMode_PosTrq;

m_IKSuccess:=FALSE;
m_targetJntPos:=m_cmdJntPos;

// update commands to arm
copyCmds(r_masterArmCtrlCmd);
END_METHOD

// calculate command wrist joint position with an optimized posture
(*wristDH=[   -deg90  a4  q4      d4;
            deg90   0   q5      0;
            -deg90  0   q6      0;
            deg90   0   q7      0];*)
// set q6 = -pi/2 for desired posture
(* wristRot = 
[ COS(q7)*SIN(q4) - COS(q4)*SIN(q5)*SIN(q7), - SIN(q4)*SIN(q7) - COS(q4)*COS(q7)*SIN(q5), -COS(q4)*COS(q5)]
[                           cos(q5)*sin(q7),                             cos(q5)*cos(q7),         -sin(q5)]
[ cos(q4)*cos(q7) + sin(q4)*sin(q5)*sin(q7),   cos(q7)*sin(q4)*sin(q5) - cos(q4)*sin(q7),  cos(q5)*sin(q4)]
*)
METHOD PROTECTED leftWristOptIK : BOOL
VAR_IN_OUT CONSTANT
	i_cmdRot :Mat3d;
END_VAR
VAR_OUTPUT
	q4 :LREAL;
	q5 :LREAL;
	q6 :LREAL;
	q7 :LREAL;
END_VAR

VAR
	q51,q52 :LREAL;
	s4,c4,s5,c5,s7,c7:LREAL;
	q4UnreachPosMin: LREAL :=-pi/2;
	q4UnreachPosMax: LREAL :=45*g_deg2Rad;
	
END_VAR
q6:=-PI/2;
// q5 = [pi-135deg, pi+135deg]
q5 := ASIN(-i_cmdRot[2,3]);
q5:= PI-q5;

// q5=3pi/2 or q5=pi/2
IF ABS(q5-3*PI/2)<g_smallAng OR ABS(q5-PI/2)<g_smallAng THEN
	q4:= -pi;
	s7:= -i_cmdRot[1,1]/(COS(q4)*SIN(q5));
	c7:= i_cmdRot[3,1]/COS(q4);
	q7:=atan2(s7,c7);
	leftWristOptIK:=TRUE;
	RETURN;
END_IF

// solution one 
c5 :=COS(q5);
s7:=i_cmdRot[2,1]/c5;
c7:= i_cmdRot[2,2]/c5;
q7:=atan2(s7,c7);

//q4=[-pi/2-225deg, -pi/2]
c4 := -i_cmdRot[1,3]/c5;
s4:= i_cmdRot[3,3]/c5;
q4:=atan2(s4,c4);
IF q4> GVL_ArmJointParameters.g_minJntPos[1,4] AND q4<GVL_ArmJointParameters.g_maxJntPos[1,4] THEN
	leftWristOptIK:=TRUE;
	RETURN;
ELSIF q4> GVL_ArmJointParameters.g_maxJntPos[1,4] AND q4-2*pi> GVL_ArmJointParameters.g_minJntPos[1,4] THEN
	q4:=q4-2*PI;
	leftWristOptIK:=TRUE;
	RETURN;
END_IF

// solution2
IF q5 > pi THEN
	q5 := 3*PI-q5;
ELSE
	q5:= pi-q5;
END_IF
IF q5 > GVL_ArmJointParameters.g_maxJntPos[1,5] OR q5<GVL_ArmJointParameters.g_minJntPos[1,5] THEN
	leftWristOptIK:=FALSE;
	RETURN;
END_IF

c5 :=COS(q5);
s7:=i_cmdRot[2,1]/c5;
c7:= i_cmdRot[2,2]/c5;
q7:=atan2(s7,c7);

c4 := -i_cmdRot[1,3]/c5;
s4:= i_cmdRot[3,3]/c5;
q4:=atan2(s4,c4);
IF q4> GVL_ArmJointParameters.g_minJntPos[1,4] AND q4<GVL_ArmJointParameters.g_maxJntPos[1,4] THEN
	leftWristOptIK:=TRUE;
	RETURN;
ELSIF q4> GVL_ArmJointParameters.g_maxJntPos[1,4] AND q4-2*pi< GVL_ArmJointParameters.g_minJntPos[1,4] THEN
	q4:=q4-2*PI;
	leftWristOptIK:=TRUE;
	RETURN;
END_IF
END_METHOD

// calculate command wrist joint position with an optimized posture
(*wristDH=[   -deg90  a4  q4      d4;
            deg90   0   q5      0;
            -deg90  0   q6      0;
            deg90   0   q7      0];*)
// set q6 = pi/2 for desired posture
(* wristRot = 
[ - cos(q7)*sin(q4) - cos(q4)*sin(q5)*sin(q7), sin(q4)*sin(q7) - cos(q4)*cos(q7)*sin(q5),  cos(q4)*cos(q5)]
[                             cos(q5)*sin(q7),                           cos(q5)*cos(q7),          sin(q5)]
[   sin(q4)*sin(q5)*sin(q7) - cos(q4)*cos(q7), cos(q4)*sin(q7) + cos(q7)*sin(q4)*sin(q5), -cos(q5)*sin(q4)]
 
*)
METHOD PROTECTED rightWristOptIK : BOOL
VAR_IN_OUT CONSTANT
	i_cmdRot :Mat3d;
END_VAR
VAR_OUTPUT
	q4 :LREAL;
	q5 :LREAL;
	q6 :LREAL;
	q7 :LREAL;
END_VAR

VAR
	q51,q52 :LREAL;
	s4,c4,s5,c5,s7,c7:LREAL;
	q4UnreachPosMin: LREAL :=-pi/2;
	q4UnreachPosMax: LREAL :=45*g_deg2Rad;
	
END_VAR
q6:=PI/2;
// q5 = [pi-135deg, pi+135deg]
q5 := ASIN(i_cmdRot[2,3]);
q5:= PI-q5;

// q5=3pi/2 or q5=pi/2
IF ABS(q5-3*PI/2)<g_smallAng OR ABS(q5-PI/2)<g_smallAng THEN
	q4:= 0;
	s7:= -i_cmdRot[1,1]/(COS(q4)*SIN(q5));
	c7:= -i_cmdRot[3,1]/COS(q4);
	q7:=atan2(s7,c7);
	rightWristOptIK:=TRUE;
	RETURN;
END_IF

// solution one 
c5 :=COS(q5);
s7:=i_cmdRot[2,1]/c5;
c7:= i_cmdRot[2,2]/c5;
q7:=atan2(s7,c7);

//q4=[-pi/2, -pi/2+225deg]
c4 := i_cmdRot[1,3]/c5;
s4:= -i_cmdRot[3,3]/c5;
q4:=atan2(s4,c4);
IF q4> GVL_ArmJointParameters.g_minJntPos[2,4] AND q4<GVL_ArmJointParameters.g_maxJntPos[2,4] THEN
	rightWristOptIK:=TRUE;
	RETURN;
END_IF

// solution2
IF q5 > pi THEN
	q5 := 3*PI-q5;
ELSE
	q5:= pi-q5;
END_IF
IF q5 > GVL_ArmJointParameters.g_maxJntPos[1,5] OR q5<GVL_ArmJointParameters.g_minJntPos[1,5] THEN
	rightWristOptIK:=FALSE;
	RETURN;
END_IF

c5 :=COS(q5);
s7:=i_cmdRot[2,1]/c5;
c7:= i_cmdRot[2,2]/c5;
q7:=atan2(s7,c7);

//q4=[-pi/2, -pi/2+225deg]
c4 := i_cmdRot[1,3]/c5;
s4:= -i_cmdRot[3,3]/c5;
q4:=atan2(s4,c4);
IF q4> GVL_ArmJointParameters.g_minJntPos[2,4] AND q4<GVL_ArmJointParameters.g_maxJntPos[2,4] THEN
	rightWristOptIK:=TRUE;
	RETURN;
END_IF
END_METHOD

METHOD PROTECTED rollFlipHandle : BOOL
VAR_INPUT
	i_armIdx:INT;
	i_curJntPos7 :LREAL;
	i_initCmdJntPos7 :LREAL;
END_VAR
VAR_OUTPUT
	o_cmdJntPos7 :LREAL;
END_VAR

VAR
	solFeasible1,solFeasible2 :BOOL;
	solIdx :INT:=0;
	halfcycleNum1, halfcycleNum2:INT;
	solution1, solution2 :LREAL;
END_VAR
// this part is used to drive gripper back near center, in case that gripper roll is stuck near limit
// TODO: remove after gripper roll has infinite motion range
IF NOT (MasterArmControl.m_masterInputDataPool.m_cartStatus.m_surgonReady) THEN
	o_cmdJntPos7:=i_initCmdJntPos7;
	rollFlipHandle:=FALSE;
	RETURN;
END_IF

// handle multiple cycles of joint7
// find the first solution within pi from current position
halfcycleNum1 := LREAL_TO_INT((i_curJntPos7 - i_initCmdJntPos7)/pi);
solution1 := halfcycleNum1 * pi + i_initCmdJntPos7;

// solution2
IF solution1 > i_curJntPos7 THEN
	solution2 := solution1 - PI;
	halfcycleNum2 := halfcycleNum1 - 1;
ELSE
	solution2 := solution1 + PI;
	halfcycleNum2 := halfcycleNum1 + 1;
END_IF

//choose the solution which is closer to current q7 which can achive orientation match with a max pi/2 degree
// NOTE: There maybe risk this joint7 is stuck at limit, which can be solved after joint7 has infinite rotation angle,
solFeasible1:=solution1> GVL_ArmJointParameters.g_minJntPos[i_armIdx,7] AND solution1< GVL_ArmJointParameters.g_maxJntPos[i_armIdx,7];
solFeasible2:=solution2> GVL_ArmJointParameters.g_minJntPos[i_armIdx,7] AND solution2< GVL_ArmJointParameters.g_maxJntPos[i_armIdx,7];
IF solFeasible1 AND solFeasible2 THEN
	IF ABS(solution1-i_curJntPos7) < ABS(solution2-i_curJntPos7)  THEN
		solIdx:=1;
	ELSE
		solIdx:=2;
	END_IF
ELSIF solFeasible1 AND NOT(solFeasible2) THEN
	solIdx:=1;
ELSIF solFeasible2 AND NOT(solFeasible1) THEN
	solIdx:=2;
ELSE
	solIdx:=0;
END_IF

IF solIdx = 1 THEN
	o_cmdJntPos7 := solution1;
	rollFlipHandle:= ((ABS(halfcycleNum1) MOD 2) = 1);
ELSIF solIdx =2 THEN
	o_cmdJntPos7 := solution2;
	rollFlipHandle:= ((ABS(halfcycleNum2) MOD 2) = 1);
ELSE
	o_cmdJntPos7:=i_initCmdJntPos7;
	rollFlipHandle:=FALSE;
END_IF
END_METHOD

// calculate position of joint 5/6/7 
(*wristDH=[   deg90   0   q5      0;
            -deg90  0   q6      0;
            deg90   0   q7      0];*)
(* wristRot = 
[ cos(q5)*cos(q6)*cos(q7) - sin(q5)*sin(q7), - cos(q7)*sin(q5) - cos(q5)*cos(q6)*sin(q7), cos(q5)*sin(q6)]
[                           cos(q7)*sin(q6),                            -sin(q6)*sin(q7),        -cos(q6)]
[ cos(q5)*sin(q7) + cos(q6)*cos(q7)*sin(q5),   cos(q5)*cos(q7) - cos(q6)*sin(q5)*sin(q7), sin(q5)*sin(q6)]
*)
METHOD PROTECTED wristIK : BOOL
VAR_IN_OUT CONSTANT
	i_cmdRot :Mat3d;
	i_masterArm :FB_MasterArm;
END_VAR

VAR_OUTPUT
	q5:	LREAL;
	q6:	LREAL;
	q7:	LREAL;
END_VAR

VAR
	invRot :Mat3d;
	jnt4Rotation :Mat3d;
	s5, s7, c5, c7:LREAL;
END_VAR
// calculate wrist joint position
// q6=[-pi/2-45deg, -pi/2+45deg]
IF 1 = i_masterArm.armIdx THEN
	q6:= -ACOS(-i_cmdRot[2,3]);
// q6=[pi/2-45deg, pi/2+45deg]
ELSE
	q6:= ACOS(-i_cmdRot[2,3]);
END_IF

IF q6>GVL_ArmJointParameters.g_maxJntPos[i_masterArm.armIdx, 6] OR q6< GVL_ArmJointParameters.g_minJntPos[i_masterArm.armIdx, 6] THEN
	wristIK:=FALSE;
	RETURN;
END_IF

// q5 = [pi-135deg, pi+135deg]
c5 := i_cmdRot[1,3]/SIN(q6);
s5 := i_cmdRot[3,3]/SIN(q6);
q5:=atan2(s5,c5);
IF q5<GVL_ArmJointParameters.g_minJntPos[1,5] THEN
	q5:=q5+2*PI;
END_IF
IF q5>GVL_ArmJointParameters.g_maxJntPos[1,5]THEN
	wristIK:=FALSE;
	RETURN;
END_IF
c7 := i_cmdRot[2,1]/SIN(q6);
s7 := -i_cmdRot[2,2]/SIN(q6);
q7:=atan2(s7,c7);
wristIK:=true;
END_METHOD

END_FUNCTION_BLOCK

// ---- FBs_StateControllers/FB_StateCtrlMasterSlave.TcPOU
// Brief: Master Arm MasterSlave controller
FUNCTION_BLOCK PUBLIC FB_StateCtrlMasterSlave EXTENDS FB_MasterArmCtrlBase
VAR_INPUT
END_VAR
VAR_OUTPUT
END_VAR
VAR
	// joint4 controller
	m_redunJntCtrl : FB_RedunJntControl;
	
	// flag if project joint4 torque to nullspace
	m_nullspaceCtrl : BOOL :=FALSE;
	
	// boundary limit force feedback
	m_boundaryForce : FB_boundaryForceFeedback;
	
	// joint torque for master-slave error
	m_boundaryTrq :Vec7d;
	
	// friction compensation scale
	m_frictionCompScale :LREAL :=1.0;

END_VAR

// override this function in each exact controller
METHOD PROTECTED calcCmdJntPos : BOOL

VAR_IN_OUT CONSTANT
	i_slaveIdx :INT;
	i_shoulderPose :ST_Frame;
	i_masterArm :FB_MasterArm;
	i_slaveStatus :ST_SlaveStatus;
END_VAR
VAR 

END_VAR
IF i_slaveStatus.m_instruStauts[i_slaveIdx].m_type = InstruType_UltrasoundKnifeS OR 
	i_slaveStatus.m_instruStauts[i_slaveIdx].m_type = InstruType_UltrasoundKnifeU THEN
	calcCmdJntPos_USKnife(i_slaveIdx,i_shoulderPose,i_masterArm,i_slaveStatus);
ELSE
	calcCmdJntPos_BasicInstru(i_slaveIdx,i_shoulderPose,i_masterArm,i_slaveStatus);
END_IF
END_METHOD

// override this function in each exact controller
METHOD PROTECTED calcCmdJntPos_BasicInstru : BOOL

VAR_IN_OUT CONSTANT
	i_slaveIdx :INT;
	i_shoulderPose :ST_Frame;
	i_masterArm :FB_MasterArm;
	i_slaveStatus :ST_SlaveStatus;
END_VAR
VAR 

END_VAR
m_cmdJntPos:=i_masterArm.curJntPos;
m_cmdJntVel:=i_masterArm.curJntVel;
m_cmdCartPose:=i_masterArm.curCartPose;
END_METHOD

// override this function in each exact controller
METHOD PROTECTED calcCmdJntPos_USKnife : BOOL

VAR_IN_OUT CONSTANT
	i_slaveIdx :INT;
	i_shoulderPose :ST_Frame;
	i_masterArm :FB_MasterArm;
	i_slaveStatus :ST_SlaveStatus;
END_VAR
VAR CONSTANT
	// orientation tracking parameters
	m_rotTrackKp : LREAL := 200;
	m_maxTrackVel :LREAL := PI;
	m_trackAngThres :LREAL := 2* g_deg2rad;
END_VAR
VAR 
	cartTrackVel :Vec3d;
	i,j : INT;
	invRot :Mat3d;
	cmdRotInView:Mat3d;
	rotT,rotErr :Mat3d;
	angle:LREAL;
	axis:Vec3d;
	
	oriJaco:Mat34;
	oriJt:Mat43;
	oriJJt:Mat3d;
	oriJJtInv:Mat3d;
	oriJPinv:Mat43;
	jntTrackVel:Vec4d;
	JpinvJ, nullJ:Mat4d;
	eye4d :Mat4d := g_eye4d;
	redunCtrlVel :Vec4d;
	jnt4TrackVel :LREAL;
	cmdZAxis, curZAxis :Vec3d;
END_VAR
m_jntOPMode[1] := DriverOPMode_Trq;
m_jntOPMode[2] := DriverOPMode_Trq;
m_jntOPMode[3] := DriverOPMode_Trq;
m_jntOPMode[4] := DriverOPMode_PosTrq;
m_jntOPMode[5] := DriverOPMode_PosTrq;
m_jntOPMode[6] := DriverOPMode_PosTrq;
m_jntOPMode[7] := DriverOPMode_Trq;

// use matched slave arm orientation as target, 
//	and transform from view coordinate to arm coordinate 
cmdRotInView := i_slaveStatus.m_curArmPose[i_slaveIdx].m_rot;
matTranspose(i_shoulderPose.m_rot, invRot);
matMultiply(invRot, cmdRotInView, m_cmdCartPose.m_rot);
m_cmdCartPose.m_pos:= i_masterArm.curCartPose.m_pos;

// first three joints and joint7 is passive control
FOR i:=1 TO 3 DO 
	m_cmdJntPos[i]:=i_masterArm.curJntPos[i];
	m_cmdJntVel[i]:=i_masterArm.curJntVel[i];
END_FOR
m_cmdJntPos[7]:=i_masterArm.curJntPos[7];
m_cmdJntVel[7]:=i_masterArm.curJntVel[7];

// compute cartesian tracking velocity
FOR i:=1 TO 3 DO
	cmdZAxis[i] :=  m_cmdCartPose.m_rot[i,3];
	curZAxis[i] := i_masterArm.simCartPose.m_rot[i,3];
END_FOR
angle := ACOS(LIMIT(-1,vecDot(cmdZAxis,curZAxis),1));
axis := cross(curZAxis, cmdZAxis);
IF ABS(angle)> g_smallAng AND ABS(angle-pi)> g_smallAng THEN
	normalize(axis);
END_IF
vecMultiNum(axis, LIMIT(-m_maxTrackVel, angle*m_rotTrackKp, m_maxTrackVel), cartTrackVel);

// compute pinv of orientation jacobian
FOR i:=1 TO 3 DO
	FOR j:=1 TO 4 DO
		oriJaco[i,j]:=i_masterArm.simJaco[i+3,j+3];
	END_FOR
END_FOR
matTranspose(oriJaco, oriJt);
matMultiply(oriJaco ,oriJt , oriJJt);
invMat3(oriJJt, oriJJtInv);
matMultiply(oriJt, oriJJtInv, oriJPinv);
matMultiVec(oriJpinv, cartTrackVel, jntTrackVel);

// calculate nullspace
matMultiply(oriJPinv, oriJaco, JpinvJ);
matSub(eye4d , JpinvJ, nullJ);

// redundant velocity
jnt4TrackVel:=calcRedunVel(i_masterArm);
redunCtrlVel[1]:=nullJ[1,1]*jnt4TrackVel;
redunCtrlVel[2]:=nullJ[2,1]*jnt4TrackVel;
redunCtrlVel[3]:=nullJ[3,1]*jnt4TrackVel;
redunCtrlVel[4]:=nullJ[4,1]*jnt4TrackVel;

// update final command joint position and velocity
FOR i :=1 TO 3 DO 
	m_cmdJntVel[i+3]:=jntTrackVel[i]+redunCtrlVel[i];
	m_cmdJntPos[i+3]:=m_cmdJntPos[i+3]+m_cmdJntVel[i+3]*g_armCtrlCycleTime;
END_FOR
END_METHOD

// override this function in each exact controller
METHOD PROTECTED calcCmdJntTrq : BOOL

VAR_IN_OUT CONSTANT
	i_slaveIdx :INT;
	i_shoulderPose :ST_Frame;
	i_masterArm :FB_MasterArm;
	i_slaveStatus :ST_SlaveStatus;
END_VAR

VAR 
	
END_VAR
IF i_slaveStatus.m_instruStauts[i_slaveIdx].m_type = InstruType_UltrasoundKnifeS OR 
	i_slaveStatus.m_instruStauts[i_slaveIdx].m_type = InstruType_UltrasoundKnifeU THEN
	calcCmdJntTrq_USKnife(i_slaveIdx,i_shoulderPose,i_masterArm,i_slaveStatus);
ELSE
	calcCmdJntTrq_BasicInstru(i_slaveIdx,i_shoulderPose,i_masterArm,i_slaveStatus);
END_IF
END_METHOD

// override this function in each exact controller
METHOD PROTECTED calcCmdJntTrq_BasicInstru : BOOL

VAR_IN_OUT CONSTANT
	i_slaveIdx :INT;
	i_shoulderPose :ST_Frame;
	i_masterArm :FB_MasterArm;
	i_slaveStatus :ST_SlaveStatus;
END_VAR

VAR 
	nullspaceMat :Mat7d;
	ctrlTrq : Vec7d;
	boundaryTrq :Vec7d;
	withinBoundary :BOOL;
	i :INT;
	inertiaTrq:LREAL;
END_VAR
// boundary force feedback
m_boundaryTrq :=m_boundaryForce.run(i_slaveIdx, i_shoulderPose, i_masterArm, i_slaveStatus);
withinBoundary := (norm(m_boundaryTrq)<g_smallNum);

// redundant joint4 controller
ctrlTrq := g_zeroVec7d;
ctrlTrq[4] := m_redunJntCtrl.run(i_masterArm, i_followEnable:=withinBoundary);

// project to nullspace
IF m_nullspaceCtrl THEN
	nullspaceMat:=i_masterArm.dynaNullspace;
	matMultiVec(nullspaceMat,ctrlTrq, m_cmdJntTrq);
	vecSelfMultiNum(m_cmdJntTrq, ctrlTrq[4] / m_cmdJntTrq[4]);
ELSE
	m_cmdJntTrq := ctrlTrq;
END_IF

// add friction compensation
FOR i:=1 TO g_mJntNum DO 
	m_cmdJntTrq[i] := m_cmdJntTrq[i] +m_frictionCompScale * i_masterArm.jntFriction[i] + m_boundaryTrq[i]+i_masterArm.jntExtTrq[i];
END_FOR
END_METHOD

// override this function in each exact controller
METHOD PROTECTED calcCmdJntTrq_USKnife : BOOL

VAR_IN_OUT CONSTANT
	i_slaveIdx :INT;
	i_shoulderPose :ST_Frame;
	i_masterArm :FB_MasterArm;
	i_slaveStatus :ST_SlaveStatus;
END_VAR

VAR 
	i :INT;
END_VAR
m_cmdJntTrq :=g_zeroVec7d;
// boundary force feedback
m_boundaryTrq :=m_boundaryForce.run(i_slaveIdx, i_shoulderPose, i_masterArm, i_slaveStatus);
m_cmdJntTrq[7] := m_boundaryTrq[7];
END_METHOD

METHOD PROTECTED calcRedunVel : LREAL
VAR_IN_OUT CONSTANT
	i_masterArm :FB_MasterArm;
END_VAR

VAR 
	// redundant control parameters
	m_jnt4AdjustKp : LREAL :=10;
	m_jnt4MaxVel :LREAL :=pi/3 ;
	m_linearVelLb :LREAL := 0.02;
	m_linearVelUb :LREAL :=0.1;	
	
	j6Bias,j5Bias :LREAL;
	velScale :LREAL;
	linearVel :Vec3d;
	curJntPos : Vec7d;
	jnt4LinkPos :LREAL;
END_VAR
// compute desired joint4 link position
curJntPos :=  i_masterArm.cmdJntPos;
jnt4LinkPos:=i_masterArm.jnt4MotorToLink(curJntPos[2],curJntPos[3],curJntPos[4]);
IF 1= i_masterArm.armIdx THEN
	j6Bias :=curJntPos[6]+PI/2;
ELSE 
	j6Bias := curJntPos[6]-PI/2;
END_IF

// scale based on joint5 position
j5Bias :=  LIMIT (0, ABS(curJntPos[5] -pi), pi/2);
j6Bias := j6Bias * ABS(COS(j5Bias));

// scale based on linear velocity
linearVel[1]:=i_masterArm.curCartTwist[1];
linearVel[2]:=i_masterArm.curCartTwist[2];
linearVel[3]:=i_masterArm.curCartTwist[3];
velScale :=LIMIT(0, (norm(linearVel)-m_linearVelLb)/(m_linearVelUb-m_linearVelLb),1.0);


calcRedunVel := LIMIT(-m_jnt4MaxVel, -j6Bias * m_jnt4AdjustKp * velScale ,m_jnt4MaxVel);

// joint limit
IF (calcRedunVel > 0 AND jnt4LinkPos+calcRedunVel * g_armCtrlCycleTime > GVL_ArmJointParameters.g_maxJntPos[i_masterArm.armIdx,4])
	 OR ( calcRedunVel <0 AND  jnt4LinkPos +calcRedunVel * g_armCtrlCycleTime< GVL_ArmJointParameters.g_minJntPos[i_masterArm.armIdx,4]) THEN
	 calcRedunVel :=0;
END_IF
END_METHOD

METHOD PUBLIC init : BOOL
VAR_IN_OUT CONSTANT
	i_masterArm	:FB_MasterArm;
END_VAR
VAR_IN_OUT 
	r_masterArmCtrlCmd :ST_ArmCtrlCmds;
END_VAR

VAR
	i:INT;
END_VAR
SUPER^.Init(i_masterArm,r_masterArmCtrlCmd);

m_jntOPMode := g_allTrqMode;
//m_jntOPMode := g_allPosMode;

// init controller
m_redunJntCtrl.init(i_masterArm);

// update commands to arm
copyCmds(r_masterArmCtrlCmd);
END_METHOD

END_FUNCTION_BLOCK

// ---- FBs_StateControllers/FB_StateCtrlGraCali.TcPOU
// Brief: Master Arm Home Posture
FUNCTION_BLOCK PUBLIC FB_StateCtrlGraCali EXTENDS FB_MasterArmCtrlBase
VAR_INPUT
END_VAR
VAR_OUTPUT
END_VAR
VAR CONSTANT
	m_caliMotionSegs :INT :=18;	
END_VAR
VAR
	// cali trajectory
	m_leftGraCaliTraj :ARRAY [1..m_caliMotionSegs, 1..g_mJntNum] OF LREAL:=
		// joint6
		[0,  -90*g_deg2Rad,    0.0,  -180*g_deg2Rad,  90*g_deg2rad,  -50*g_deg2rad, 0.0 , 
		 0, -90*g_deg2rad,   0.0,  -180*g_deg2rad,   90*g_deg2rad,  -130*g_deg2rad,  0,
		 0,  -90*g_deg2Rad,    0.0,  -180*g_deg2Rad,  90*g_deg2rad,  -50*g_deg2rad, 0.0 , 
		// joint5
		 0.0,  -90*g_deg2Rad,   0*g_deg2Rad,  -180*g_deg2Rad,  90*g_deg2Rad,  -90*g_deg2Rad,    0,
		 0.0,  -90*g_deg2Rad,  0*g_deg2Rad, -180*g_deg2Rad,  270*g_deg2Rad,  -90*g_deg2Rad,     0,
		0.0,  -90*g_deg2Rad,   0*g_deg2Rad,  -180*g_deg2Rad,  90*g_deg2Rad,  -90*g_deg2Rad,    0,
		// joint4
		 0.0,  -90*g_deg2Rad,   -30*g_deg2Rad,  -150*g_deg2Rad,  180*g_deg2Rad,  -90*g_deg2Rad,    0,
		 0.0,  -90*g_deg2Rad,  -30*g_deg2Rad, -210*g_deg2Rad,  180*g_deg2Rad,  -90*g_deg2Rad,     0,
		0.0,  -90*g_deg2Rad,   -30*g_deg2Rad,  -150*g_deg2Rad,  180*g_deg2Rad,  -90*g_deg2Rad,    0,
		// joint3
		 0.0,  -90*g_deg2Rad,   -30*g_deg2Rad,  -180*g_deg2Rad,  180*g_deg2Rad,  -90*g_deg2Rad,    0,
		 0.0,  -90*g_deg2Rad,  30*g_deg2Rad, -180*g_deg2Rad,  180*g_deg2Rad,  -90*g_deg2Rad,     0,
		0.0,  -90*g_deg2Rad,   -30*g_deg2Rad,  -180*g_deg2Rad,  180*g_deg2Rad,  -90*g_deg2Rad,    0,
		// joint2
		 0.0,  -75*g_deg2Rad,   0*g_deg2Rad,  -180*g_deg2Rad,  180*g_deg2Rad,  -90*g_deg2Rad,    0,
		 0.0,  -120*g_deg2Rad,  0*g_deg2Rad, -180*g_deg2Rad,  180*g_deg2Rad,  -90*g_deg2Rad,     0,
		0.0,  -75*g_deg2Rad,   0*g_deg2Rad,  -180*g_deg2Rad,  180*g_deg2Rad,  -90*g_deg2Rad,    0,
		// joint1/7
		 0.0*g_deg2Rad,  -90*g_deg2Rad,   0*g_deg2Rad,  -180*g_deg2Rad,  180*g_deg2Rad,  -90*g_deg2Rad,    45*g_deg2Rad,
		 -30.0*g_deg2Rad,  -90*g_deg2Rad,  0*g_deg2Rad, -180*g_deg2Rad,  180*g_deg2Rad,  -90*g_deg2Rad,     -45*g_deg2Rad,
		0.0*g_deg2Rad,  -90*g_deg2Rad,   0*g_deg2Rad,  -180*g_deg2Rad,  180*g_deg2Rad,  -90*g_deg2Rad,    45*g_deg2Rad];
		
	m_rightGraCaliTraj :ARRAY [1..m_caliMotionSegs, 1..g_mJntNum] OF LREAL:=
		// joint6
		[0,  -90*g_deg2Rad,    0.0,  0*g_deg2Rad,  270*g_deg2rad,  50*g_deg2rad, 0.0 , 
		 0, -90*g_deg2rad,   0.0,  0*g_deg2rad,   270*g_deg2rad,  130*g_deg2rad,  0,
		 0,  -90*g_deg2Rad,    0.0,  0*g_deg2Rad,  270*g_deg2rad,  50*g_deg2rad, 0.0 , 
		// joint5
		 0.0,  -90*g_deg2Rad,   0*g_deg2Rad,  0*g_deg2Rad,  270*g_deg2Rad,  90*g_deg2Rad,    0,
		 0.0,  -90*g_deg2Rad,  0*g_deg2Rad, 0*g_deg2Rad,  90*g_deg2Rad,  90*g_deg2Rad,     0,
		0.0,  -90*g_deg2Rad,   0*g_deg2Rad,  0*g_deg2Rad,  270*g_deg2Rad,  90*g_deg2Rad,    0,
		// joint4
		 0.0,  -90*g_deg2Rad,   -30*g_deg2Rad,  30*g_deg2Rad,  180*g_deg2Rad,  90*g_deg2Rad,    0,
		 0.0,  -90*g_deg2Rad,  -30*g_deg2Rad, -30*g_deg2Rad,  180*g_deg2Rad,  90*g_deg2Rad,     0,
		0.0,  -90*g_deg2Rad,   -30*g_deg2Rad,  30*g_deg2Rad,  180*g_deg2Rad,  90*g_deg2Rad,    0,
		// joint3
		 0.0,  -90*g_deg2Rad,   -30*g_deg2Rad,  0*g_deg2Rad,  180*g_deg2Rad,  90*g_deg2Rad,    0,
		 0.0,  -90*g_deg2Rad,  30*g_deg2Rad, 0*g_deg2Rad,  180*g_deg2Rad,  90*g_deg2Rad,     0,
		0.0,  -90*g_deg2Rad,   -30*g_deg2Rad,  0*g_deg2Rad,  180*g_deg2Rad,  90*g_deg2Rad,    0,
		// joint2
		 0.0,  -75*g_deg2Rad,   0*g_deg2Rad,  0*g_deg2Rad,  180*g_deg2Rad,  90*g_deg2Rad,    0,
		 0.0,  -120*g_deg2Rad,  0*g_deg2Rad, 0*g_deg2Rad,  180*g_deg2Rad,  90*g_deg2Rad,     0,
		0.0,  -75*g_deg2Rad,   0*g_deg2Rad,  0*g_deg2Rad,  180*g_deg2Rad,  90*g_deg2Rad,    0,
		// joint1/7
		 0.0*g_deg2Rad,  -90*g_deg2Rad,   0*g_deg2Rad,  0*g_deg2Rad,  180*g_deg2Rad,  90*g_deg2Rad,    45*g_deg2Rad,
		 30.0*g_deg2Rad,  -90*g_deg2Rad,  0*g_deg2Rad, 0*g_deg2Rad,  180*g_deg2Rad,  90*g_deg2Rad,     -45*g_deg2Rad,
		0.0*g_deg2Rad,  -90*g_deg2Rad,   0*g_deg2Rad,  0*g_deg2Rad,  180*g_deg2Rad,  90*g_deg2Rad,    45*g_deg2Rad];
		
	

	m_transMaxjntVel:Vec7d:=[7(30*g_deg2rad)];
	m_caliMaxjntVel:Vec7d:=[7(5.0*g_deg2rad)];
	m_caliMaxjntAcc:Vec7d:=[7(1.0)];
	m_caliMaxjntJerk:Vec7d:=[7(2.0)];
	
	m_caliTrajIdx: INT := 1;
	m_caliPlanner: ARRAY[1..m_caliMotionSegs] OF FB_TrajMoveJ;
	
	
END_VAR

// override this function in each exact controller
METHOD PROTECTED calcCmdJntPos : BOOL

VAR_IN_OUT CONSTANT
	i_slaveIdx :INT;
	i_shoulderPose :ST_Frame;
	i_masterArm :FB_MasterArm;
	i_slaveStatus :ST_SlaveStatus;
END_VAR
VAR 
	i :INT;
	curJntVel :Vec7d;
END_VAR
// check if planner is ready
IF m_caliPlanner[m_caliTrajIdx].isGene = FALSE THEN
	calcCmdJntPos:=FALSE;
	RETURN;
END_IF

// traj plan
calcCmdJntPos :=m_caliPlanner[m_caliTrajIdx].evaluate(m_timePeriod, jntPos=> m_cmdJntPos, jntVel=>m_cmdJntVel, jntAcc=> m_cmdJntAcc);

// check if to transit to next segment
curJntVel :=i_masterArm.curJntVel;
IF(m_timePeriod > m_caliPlanner[m_caliTrajIdx].duration  AND norm(curJntVel)<7*g_jntStaticVelThres) THEN
	m_caliTrajIdx:=m_caliTrajIdx+1;
	m_timePeriod:=0;
END_IF

// check if to terminated
IF(m_caliTrajIdx > m_caliMotionSegs) THEN
	m_isFinished:=TRUE;
END_IF
END_METHOD

METHOD PUBLIC init : BOOL
VAR_IN_OUT CONSTANT
	i_masterArm	:FB_MasterArm;
END_VAR
VAR_IN_OUT 
	r_masterArmCtrlCmd :ST_ArmCtrlCmds;
END_VAR

VAR
	i,j :INT;
	startJntPos,endJntPos ,maxVel :Vec7d;
	
	
	
END_VAR
SUPER^.Init(i_masterArm,r_masterArmCtrlCmd);
m_caliTrajIdx :=1;

FOR i:=1 TO m_caliMotionSegs DO
	IF (i mod 3) = 1 THEN
		maxVel := m_transMaxjntVel;
	ELSE
		maxVel := m_caliMaxjntVel;
	END_IF
	
	IF i_masterArm.armIdx=1 THEN
		FOR j:=1 TO 7 DO 
			endJntPos[j]:=m_leftGraCaliTraj[i,j];
			IF i =1 THEN
				startJntPos[j]:=i_masterArm.curJntPos[j];
			ELSE
				startJntPos[j]:=m_leftGraCaliTraj[i-1,j];
			END_IF
		END_FOR
	ELSE
		FOR j:=1 TO 7 DO 
			endJntPos[j]:=m_rightGraCaliTraj[i,j];
			IF i =1 THEN
				startJntPos[j]:=i_masterArm.curJntPos[j];
			ELSE
				startJntPos[j]:=m_rightGraCaliTraj[i-1,j];
			END_IF
		END_FOR
	END_IF
	
	m_caliPlanner[i].init(startJntPos,endJntPos,maxVel, m_caliMaxJntAcc, m_caliMaxJntAcc);
END_FOR


// update commands to arm
copyCmds(r_masterArmCtrlCmd);
END_METHOD

END_FUNCTION_BLOCK

// ---- FBs_StateControllers/FB_StateCtrlTest.TcPOU
// Brief: Master Arm Test
FUNCTION_BLOCK PUBLIC FB_StateCtrlTest EXTENDS FB_MasterArmCtrlBase
VAR_INPUT
END_VAR
VAR_OUTPUT
END_VAR
VAR
	// ################ variables for single DH  joint test ##################
	m_freqTestFlag :BOOL:=FALSE;
	m_initJntPos :Vec7d;
	m_jntMotionFreq :Vec7d :=[0.2, 0.2, 0.1, 4(0.1)];
	m_jntMotionRange :Vec7d :=[pi/6, pi/6, 0.1, 4(pi/6)];
	m_testJntIdx :INT :=1;
	
	m_stepTestFlag :BOOL :=FALSE;
	m_jntStep : LREAL := 0*g_deg2Rad;
	
END_VAR

METHOD PROTECTED calcCmdJntPos : BOOL
VAR_IN_OUT CONSTANT
	i_slaveIdx :INT;
	i_shoulderPose :ST_Frame;
	i_masterArm :FB_MasterArm;
	i_slaveStatus :ST_SlaveStatus;
END_VAR

VAR 
	errThres :LREAL;
	m_masterGripAngle: INT;
END_VAR
// Just for joint controller test
IF m_testJntIdx >=1 AND m_testJntIdx <=7 THEN
	IF m_freqTestFlag THEN 
		m_cmdJntPos[m_testJntIdx]:=m_initJntPos[m_testJntIdx]+m_jntMotionRange[m_testJntIdx]/2
										+0.5*m_jntMotionRange[m_testJntIdx]*SIN(2*pi*m_jntMotionFreq[m_testJntIdx]*m_timePeriod-pi/2);
		m_cmdJntVel[m_testJntIdx]:=0.5*m_jntMotionRange[m_testJntIdx]*2*pi*m_jntMotionFreq[m_testJntIdx]*COS(2*pi*m_jntMotionFreq[m_testJntIdx]*m_timePeriod-pi/2);
	ELSIF m_stepTestFlag THEN
		m_cmdJntPos[m_testJntIdx]:=m_initJntPos[m_testJntIdx]+m_jntStep;
		m_cmdJntVel[m_testJntIdx]:=0;
	ELSE
		m_timePeriod:=0;
	END_IF
	
END_IF


//FOR i:=1 TO 3 DO 
//		errThres :=5*g_deg2rad;
//	IF ABS(m_cmdJntPos[i]-i_masterArm.curJntPos[i])>errThres THEN
//		m_isFinished:=TRUE;
//	END_IF
	
//END_FOR
END_METHOD

METHOD PUBLIC init : BOOL
VAR_IN_OUT CONSTANT
	i_masterArm	:FB_MasterArm;
END_VAR
VAR_IN_OUT 
	r_masterArmCtrlCmd :ST_ArmCtrlCmds;
END_VAR
// check if to hold the command joint position unchanged
m_holdLastCmds := checkToHoldLastCmds(i_masterArm);

// init
SUPER^.Init(i_masterArm,r_masterArmCtrlCmd);

m_initJntPos := i_masterArm.curJntPos;

m_jntOPMode := g_allPosTrqMode;

// update commands to arm
copyCmds(r_masterArmCtrlCmd);
END_METHOD

END_FUNCTION_BLOCK

// ---- FBs_StateControllers/FB_StateCtrlDisable.TcPOU
// Brief: Master Arm Error Hold
FUNCTION_BLOCK PUBLIC FB_StateCtrlDisable EXTENDS FB_MasterArmCtrlBase
VAR_INPUT
END_VAR
VAR_OUTPUT
END_VAR
VAR
END_VAR

// override this function in each exact controller
METHOD PROTECTED calcCmdJntPos : BOOL

VAR_IN_OUT CONSTANT
	i_slaveIdx :INT;
	i_shoulderPose :ST_Frame;
	i_masterArm :FB_MasterArm;
	i_slaveStatus :ST_SlaveStatus;
END_VAR
var 
	i,j : INT;

	
END_VAR
m_cmdJntPos:= i_masterArm.curJntPos;
m_cmdJntVel := g_zeroVec7d;
END_METHOD

METHOD PUBLIC init : BOOL
VAR_IN_OUT CONSTANT
	i_masterArm	:FB_MasterArm;
END_VAR
VAR_IN_OUT 
	r_masterArmCtrlCmd :ST_ArmCtrlCmds;
END_VAR

VAR
	i:INT;
END_VAR
SUPER^.Init(i_masterArm,r_masterArmCtrlCmd);
m_jntOPMode:=g_allPosMode;

// disable all joints
m_jntEnableFlag :=g_zeroVec7i;
END_METHOD

END_FUNCTION_BLOCK

// ---- SafetyCheck/Fb_SafetyCheck.TcPOU
FUNCTION_BLOCK Fb_SafetyCheck
VAR_INPUT
END_VAR
VAR_OUTPUT
END_VAR
VAR
	i, j:INT;
	m_checkDelay :ARRAY[1..g_maxNum] OF checkDelay;
	m_checkDelayTime :checkDelayTime;
	m_checkPermit:ARRAY[1..g_maxNum] OF  checkPermit;
	
	m_jntErrFlag:ARRAY[1..g_maxNum,0..g_maxArmJoint,1..3] OF BOOL;
	m_armErrFlag:ARRAY [1..g_maxNum,1..3] OF BOOL;
	m_errCode:UDINT;
	
	
	m_errNumType: ARRAY [1..3] OF INT;
	m_ArrayErrCodeType:ARRAY [1..3] OF ARRAY [0..100] OF UDINT;
	
	//The fault is sent to the UI at the frequency of 0.1S
	m_errCodeUpdateFlag: ARRAY [1..3] OF BOOL;
	m_errCodeUpdateTon: ARRAY [1..3] OF TON;
	
	m_curJntTorqueIOlast :ARRAY [1..g_maxArmNum] OF vec7di;  
	m_cmdJntPosLast : ARRAY [1..g_maxArmNum] OF vec7d;  
	m_cartCurJntTorqueIOlast :ARRAY [1..4] OF LREAL;  
	m_cartCmdJntPosLast : ARRAY [1..4] OF LREAL; 
	o_ErrCode:ARRAY [1..3] OF UDINT;
		
	//error robot data record
	m_dataRecord : Fb_dataRecord;
	
	m_PromptMassBusy:BOOL;
	m_PromptFlag:ARRAY[1..g_maxNum,1..20] OF UINT;
	m_deleteCode:UDINT;
	
END_VAR


VAR CONSTANT
	m_codeUpdateDelay:TIME:=T#0.1S;
	
	//Fault level: 1 indicates  prompt message, 2 indicates a recoverable fault and 3 indicates an unrecoverable fault
	m_promptMessageLevel : UINT :=1;
	m_rcvLevel : UINT :=2;
	m_unrcvLevel : UINT :=3;
END_VAR

